KUKA KRL program: MyProgram_087().src

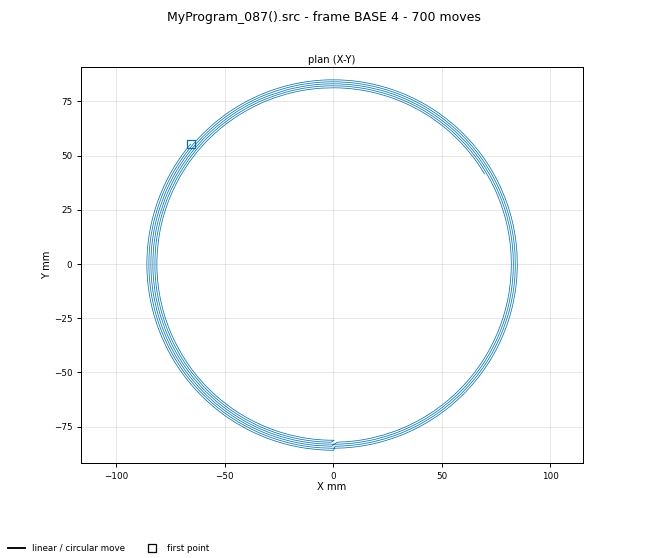
[picture p0: tool path of MyProgram_087().src in frame BASE 4, 700 of 700 moves have a stored position in this frame; points joined in program order, loops and branches not executed]
&ACCESS RVP
&REL 1
&PARAM TEMPLATE = C:\KRC\Roboter\Template\vorgabe
&PARAM EDITMASK = *
DEF MyProgram_087()
; ---- Setting reference (Base) ----
$BASE = BASE_DATA[4]

; --------------------------
; ---- Setting tool (TCP) ----
$TOOL = TOOL_DATA[3]
; --------------------------

$VEL.CP = VEL_APROX_PRINT
Startdeposition()
$VEL.CP = VEL_PRINT
LIN {X -65.6493,Y 55.3345,Z 85,A 135.0931,B 24.9031,C -2.2728,E1 24.8765,E2 309.7224} C_DIS
LIN {X -67.6092,Y 52.9216,Z 85,A 137.2051,B 24.9035,C -2.2684,E1 24.8729,E2 307.6109} C_DIS
LIN {X -69.5478,Y 50.3473,Z 85,A 139.3855,B 24.9039,C -2.2635,E1 24.8693,E2 305.4317} C_DIS
LIN {X -71.5517,Y 47.4546,Z 85,A 141.6093,B 24.9047,C -2.2535,E1 24.8658,E2 303.2206} C_DIS
LIN {X -73.3166,Y 44.6791,Z 85,A 143.8272,B 24.9052,C -2.248,E1 24.8625,E2 301.0046} C_DIS
LIN {X -75.0457,Y 41.7097,Z 85,A 146.1939,B 24.9056,C -2.2435,E1 24.8592,E2 298.6364} C_DIS
LIN {X -76.7013,Y 38.583,Z 85,A 148.5855,B 24.9061,C -2.2374,E1 24.8562,E2 296.2465} C_DIS
LIN {X -78.0463,Y 35.7848,Z 85,A 150.7651,B 24.9064,C -2.2343,E1 24.8536,E2 294.0624} C_DIS
LIN {X -79.8151,Y 31.6411,Z 85,A 154.2705,B 24.9059,C -2.2392,E1 24.8499,E2 290.5257} C_DIS
LIN {X -81.0653,Y 28.2839,Z 85,A 156.0322,B 24.908,C -2.2142,E1 24.8483,E2 288.8137} C_DIS
LIN {X -82.0788,Y 25.1926,Z 85,A 158.531,B 24.9078,C -2.2166,E1 24.8462,E2 286.2947} C_DIS
LIN {X -83.1814,Y 21.2698,Z 85,A 160.8924,B 24.9094,C -2.1981,E1 24.8445,E2 283.9638} C_DIS
LIN {X -83.8706,Y 18.3647,Z 85,A 162.9269,B 24.9098,C -2.193,E1 24.8432,E2 281.9297} C_DIS
LIN {X -84.5105,Y 15.1494,Z 85,A 165.1334,B 24.9103,C -2.1866,E1 24.8421,E2 279.7254} C_DIS
LIN {X -84.9815,Y 12.2354,Z 85,A 167.1994,B 24.9106,C -2.183,E1 24.8412,E2 277.6557} C_DIS
LIN {X -85.4194,Y 8.6682,Z 85,A 169.6631,B 24.9111,C -2.1771,E1 24.8404,E2 275.1912} C_DIS
LIN {X -85.7088,Y 5.064,Z 85,A 171.7651,B 24.9124,C -2.1608,E1 24.84,E2 273.1156} C_DIS
LIN {X -85.8246,Y 2.3935,Z 85,A 173.796,B 24.9124,C -2.1619,E1 24.8398,E2 271.0697} C_DIS
LIN {X -85.8549,Y -0.7778,Z 85,A 175.8922,B 24.9129,C -2.1546,E1 24.8398,E2 268.9783} C_DIS
LIN {X -85.7663,Y -3.9684,Z 85,A 178.1489,B 24.9132,C -2.1514,E1 24.84,E2 266.7158} C_DIS
LIN {X -85.5328,Y -7.4731,Z 85,A -179.4836,B 24.9137,C -2.1446,E1 24.8406,E2 264.3502} C_DIS
LIN {X -85.1548,Y -10.9633,Z 85,A -177.1748,B 24.9144,C -2.1363,E1 24.8413,E2 262.0474} C_DIS
LIN {X -84.6385,Y -14.4197,Z 85,A -174.7821,B 24.9149,C -2.1307,E1 24.8424,E2 259.6538} C_DIS
LIN {X -84.1506,Y -17.0373,Z 85,A -173.063,B 24.9154,C -2.1236,E1 24.8433,E2 257.9415} C_DIS
LIN {X -83.4534,Y -20.1765,Z 85,A -170.9028,B 24.9159,C -2.1175,E1 24.8447,E2 255.7833} C_DIS
LIN {X -82.61,Y -23.3907,Z 85,A -168.7117,B 24.9165,C -2.11,E1 24.8463,E2 253.5972} C_DIS
LIN {X -81.3101,Y -27.5722,Z 85,A -165.6983,B 24.917,C -2.1039,E1 24.8488,E2 250.5811} C_DIS
LIN {X -80.4535,Y -29.9829,Z 85,A -163.7906,B 24.917,C -2.1046,E1 24.8507,E2 248.6611} C_DIS
LIN {X -79.1046,Y -33.3765,Z 85,A -161.4857,B 24.9178,C -2.0939,E1 24.8531,E2 246.369} C_DIS
LIN {X -77.6498,Y -36.6364,Z 85,A -159.0613,B 24.9182,C -2.0883,E1 24.856,E2 243.9444} C_DIS
LIN {X -76.0628,Y -39.8249,Z 85,A -156.9851,B 24.9194,C -2.0733,E1 24.8585,E2 241.893} C_DIS
LIN {X -74.7201,Y -42.2926,Z 85,A -154.847,B 24.9192,C -2.0757,E1 24.8615,E2 239.7378} C_DIS
LIN {X -73.1736,Y -44.9144,Z 85,A -152.7759,B 24.9195,C -2.0716,E1 24.8645,E2 237.666} C_DIS
LIN {X -71.3839,Y -47.7089,Z 85,A -150.4876,B 24.9198,C -2.068,E1 24.868,E2 235.3747} C_DIS
LIN {X -69.3777,Y -50.5796,Z 85,A -148.2542,B 24.9205,C -2.0593,E1 24.8716,E2 233.1512} C_DIS
LIN {X -67.3565,Y -53.2413,Z 85,A -146.0514,B 24.9209,C -2.0532,E1 24.8753,E2 230.9526} C_DIS
LIN {X -65.2873,Y -55.7594,Z 85,A -143.9463,B 24.9215,C -2.0461,E1 24.8791,E2 228.8546} C_DIS
LIN {X -63.1419,Y -58.1779,Z 85,A -141.5868,B 24.9215,C -2.0472,E1 24.8835,E2 226.482} C_DIS
LIN {X -60.5197,Y -60.9013,Z 85,A -139.0966,B 24.9219,C -2.0409,E1 24.8884,E2 223.9962} C_DIS
LIN {X -58.0252,Y -63.282,Z 85,A -136.8032,B 24.9223,C -2.0361,E1 24.8931,E2 221.705} C_DIS
LIN {X -55.4826,Y -65.5232,Z 85,A -134.4958,B 24.9225,C -2.033,E1 24.8979,E2 219.3957} C_DIS
LIN {X -52.8303,Y -67.6812,Z 85,A -132.4193,B 24.9233,C -2.0228,E1 24.9024,E2 217.3358} C_DIS
LIN {X -50.6058,Y -69.3586,Z 85,A -130.3248,B 24.923,C -2.0266,E1 24.9072,E2 215.2249} C_DIS
LIN {X -47.7844,Y -71.3328,Z 85,A -128.0592,B 24.9233,C -2.0219,E1 24.9124,E2 212.9629} C_DIS
LIN {X -45.133,Y -73.0392,Z 85,A -125.8563,B 24.9233,C -2.0217,E1 24.9176,E2 210.7534} C_DIS
LIN {X -40.4274,Y -75.7455,Z 85,A -121.6598,B 24.9224,C -2.0342,E1 24.928,E2 206.5152} C_DIS
LIN {X -37.144,Y -77.4071,Z 85,A -120.0392,B 24.9246,C -2.0059,E1 24.9319,E2 204.9577} C_DIS
LIN {X -34.4456,Y -78.6451,Z 85,A -117.8993,B 24.9244,C -2.0085,E1 24.9374,E2 202.8064} C_DIS
LIN {X -31.4797,Y -79.8785,Z 85,A -115.7324,B 24.9244,C -2.0071,E1 24.943,E2 200.638} C_DIS
LIN {X -28.5704,Y -80.9647,Z 85,A -113.6156,B 24.9244,C -2.0067,E1 24.9485,E2 198.518} C_DIS
LIN {X -25.5353,Y -81.9725,Z 85,A -111.4952,B 24.9247,C -2.0046,E1 24.9542,E2 196.3986} C_DIS
LIN {X -22.9181,Y -82.7438,Z 85,A -109.595,B 24.9246,C -2.0059,E1 24.9593,E2 194.4924} C_DIS
LIN {X -19.7547,Y -83.555,Z 85,A -107.4358,B 24.9246,C -2.0041,E1 24.9651,E2 192.3345} C_DIS
LIN {X -15.6717,Y -84.4166,Z 85,A -104.7417,B 24.925,C -2.0001,E1 24.9725,E2 189.6467} C_DIS
LIN {X -12.5082,Y -84.9427,Z 85,A -102.5283,B 24.9249,C -2.0019,E1 24.9786,E2 187.4273} C_DIS
LIN {X -6.7373,Y -85.5929,Z 85,A -99.1371,B 24.926,C -1.9862,E1 24.988,E2 184.071} C_DIS
LIN {X -3.1736,Y -85.8004,Z 85,A -96.2343,B 24.9248,C -2.0028,E1 24.9962,E2 181.1283} C_DIS
LIN {X 0.2479,Y -85.8577,Z 85,A -93.4453,B 24.9235,C -2.0194,E1 25.0041,E2 178.2998} C_DIS
LIN {X 0.2479,Y -85.8577,Z 85,A -93.4453,B 24.9235,C -2.0194,E1 25.0041,E2 178.2998} C_DIS
Enddeposition()
LIN {X 0.5365,Y -84.9273,Z 85,A -93.1479,B 24.9221,C -2.0386,E1 25.005,E2 177.9569} C_DIS
Startdeposition()
$VEL.CP = VEL_PRINT
LIN {X -0.353,Y -84.9359,Z 85,A -96.7334,B 24.929,C -1.9459,E1 24.9944,E2 181.7624} C_DIS
LIN {X -5.9457,Y -84.7284,Z 85,A -99.0371,B 24.9257,C -1.9903,E1 24.9883,E2 183.9613} C_DIS
LIN {X -10.0146,Y -84.3441,Z 85,A -101.4892,B 24.925,C -1.9999,E1 24.9815,E2 186.3921} C_DIS
LIN {X -12.0876,Y -84.0721,Z 85,A -103.4806,B 24.9263,C -1.9825,E1 24.9759,E2 188.4264} C_DIS
LIN {X -15.4591,Y -83.5189,Z 85,A -105.8149,B 24.9263,C -1.9823,E1 24.9694,E2 190.7634} C_DIS
LIN {X -18.4006,Y -82.9197,Z 85,A -107.581,B 24.9257,C -1.991,E1 24.9647,E2 192.511} C_DIS
LIN {X -20.6463,Y -82.3905,Z 85,A -109.6817,B 24.9268,C -1.9755,E1 24.9589,E2 194.6514} C_DIS
LIN {X -24.6804,Y -81.2731,Z 85,A -112.2511,B 24.9261,C -1.985,E1 24.952,E2 197.2025} C_DIS
LIN {X -27.9054,Y -80.2219,Z 85,A -114.4048,B 24.9257,C -1.9908,E1 24.9464,E2 199.3464} C_DIS
LIN {X -31.5185,Y -78.8735,Z 85,A -117.0724,B 24.9257,C -1.9913,E1 24.9394,E2 202.0186} C_DIS
LIN {X -34.387,Y -77.6647,Z 85,A -119.1143,B 24.9254,C -1.9952,E1 24.9342,E2 204.0559} C_DIS
LIN {X -37.47,Y -76.2252,Z 85,A -121.8843,B 24.9262,C -1.9841,E1 24.9271,E2 206.8596} C_DIS
LIN {X -42.911,Y -73.3006,Z 85,A -125.5069,B 24.9246,C -2.0055,E1 24.9184,E2 210.4415} C_DIS
LIN {X -45.7094,Y -71.5883,Z 85,A -127.4702,B 24.9238,C -2.016,E1 24.9137,E2 212.3858} C_DIS
LIN {X -47.6622,Y -70.3031,Z 85,A -129.5782,B 24.9248,C -2.0032,E1 24.9088,E2 214.5315} C_DIS
LIN {X -50.2302,Y -68.4918,Z 85,A -131.9925,B 24.9251,C -1.9984,E1 24.9033,E2 216.9657} C_DIS
LIN {X -53.1184,Y -66.2786,Z 85,A -134.0621,B 24.924,C -2.0137,E1 24.8988,E2 219.0065} C_DIS
LIN {X -55.5704,Y -64.2362,Z 85,A -136.208,B 24.9236,C -2.018,E1 24.8942,E2 221.1505} C_DIS
LIN {X -57.9324,Y -62.1141,Z 85,A -138.3687,B 24.9234,C -2.0217,E1 24.8898,E2 223.311} C_DIS
LIN {X -60.7411,Y -59.371,Z 85,A -140.818,B 24.9225,C -2.0329,E1 24.885,E2 225.744} C_DIS
LIN {X -62.5685,Y -57.4402,Z 85,A -143.2624,B 24.9236,C -2.0185,E1 24.8802,E2 228.2333} C_DIS
LIN {X -65.9427,Y -53.5329,Z 85,A -146.2237,B 24.9219,C -2.0411,E1 24.875,E2 231.1545} C_DIS
LIN {X -67.897,Y -51.0314,Z 85,A -148.3795,B 24.9215,C -2.0458,E1 24.8713,E2 233.3093} C_DIS
LIN {X -70.6126,Y -47.2051,Z 85,A -151.4442,B 24.9207,C -2.0565,E1 24.8664,E2 236.3637} C_DIS
LIN {X -73.0277,Y -43.3726,Z 85,A -154.3157,B 24.9197,C -2.0695,E1 24.8622,E2 239.2187} C_DIS
LIN {X -74.9807,Y -39.9027,Z 85,A -157.1365,B 24.9194,C -2.0729,E1 24.8584,E2 242.0461} C_DIS
LIN {X -75.98,Y -37.9647,Z 85,A -158.8511,B 24.9196,C -2.0703,E1 24.8562,E2 243.7763} C_DIS
LIN {X -77.3687,Y -35.0474,Z 85,A -161.3363,B 24.9198,C -2.068,E1 24.8532,E2 246.2804} C_DIS
LIN {X -78.933,Y -31.3672,Z 85,A -164.1892,B 24.9195,C -2.0715,E1 24.8502,E2 249.1409} C_DIS
LIN {X -80.2911,Y -27.7072,Z 85,A -167.1343,B 24.9195,C -2.0708,E1 24.8475,E2 252.1044} C_DIS
LIN {X -81.4269,Y -24.1634,Z 85,A -168.8871,B 24.9174,C -2.0988,E1 24.8461,E2 253.8004} C_DIS
LIN {X -82.2605,Y -21.1522,Z 85,A -171.0204,B 24.9169,C -2.1045,E1 24.8446,E2 255.9326} C_DIS
LIN {X -83.1881,Y -17.1447,Z 85,A -173.9455,B 24.9166,C -2.1089,E1 24.8428,E2 258.8643} C_DIS
LIN {X -83.6593,Y -14.6784,Z 85,A -175.662,B 24.9162,C -2.1135,E1 24.8419,E2 260.58} C_DIS
LIN {X -84.1818,Y -11.3038,Z 85,A -177.9693,B 24.9157,C -2.1206,E1 24.841,E2 262.8841} C_DIS
LIN {X -84.6052,Y -7.5007,Z 85,A 179.4059,B 24.9151,C -2.1276,E1 24.8403,E2 265.508} C_DIS
LIN {X -84.7879,Y -5.034,Z 85,A 177.7703,B 24.9146,C -2.1338,E1 24.84,E2 267.1386} C_DIS
LIN {X -84.9203,Y -1.658,Z 85,A 175.5344,B 24.9139,C -2.1422,E1 24.8398,E2 269.3679} C_DIS
LIN {X -84.8865,Y 2.9297,Z 85,A 172.2129,B 24.9136,C -2.146,E1 24.84,E2 272.7004} C_DIS
LIN {X -84.6468,Y 7.0133,Z 85,A 169.6641,B 24.9125,C -2.1605,E1 24.8404,E2 275.23} C_DIS
LIN {X -84.3125,Y 10.2846,Z 85,A 167.392,B 24.912,C -2.1661,E1 24.8411,E2 277.5022} C_DIS
LIN {X -83.9048,Y 13.2,Z 85,A 165.3074,B 24.9117,C -2.1697,E1 24.842,E2 279.5905} C_DIS
LIN {X -83.0805,Y 17.6644,Z 85,A 162.5154,B 24.9103,C -2.1867,E1 24.8435,E2 282.3585} C_DIS
LIN {X -82.5476,Y 20.0028,Z 85,A 160.707,B 24.9103,C -2.1867,E1 24.8446,E2 284.1775} C_DIS
LIN {X -81.0132,Y 25.5189,Z 85,A 156.6749,B 24.9097,C -2.1942,E1 24.8478,E2 288.2152} C_DIS
LIN {X -79.098,Y 30.9471,Z 85,A 153.0309,B 24.9082,C -2.2125,E1 24.8512,E2 291.8359} C_DIS
LIN {X -78.0524,Y 33.4972,Z 85,A 150.7435,B 24.9087,C -2.2066,E1 24.8537,E2 294.1503} C_DIS
LIN {X -76.3679,Y 37.1793,Z 85,A 147.8244,B 24.9084,C -2.2096,E1 24.8572,E2 297.078} C_DIS
LIN {X -74.7656,Y 40.3033,Z 85,A 145.8649,B 24.9069,C -2.2275,E1 24.8597,E2 299.0051} C_DIS
LIN {X -73.177,Y 43.1202,Z 85,A 143.6694,B 24.9064,C -2.2334,E1 24.8628,E2 301.198} C_DIS
LIN {X -70.9482,Y 46.6965,Z 85,A 140.868,B 24.9057,C -2.2425,E1 24.867,E2 303.992} C_DIS
LIN {X -69.2232,Y 49.2176,Z 85,A 138.7614,B 24.9053,C -2.2469,E1 24.8703,E2 306.0985} C_DIS
LIN {X -67.3467,Y 51.7555,Z 85,A 136.6237,B 24.9048,C -2.2523,E1 24.8739,E2 308.2334} C_DIS
LIN {X -65.0503,Y 54.6154,Z 85,A 134.0242,B 24.9046,C -2.2553,E1 24.8785,E2 310.838} C_DIS
LIN {X -62.2698,Y 57.7639,Z 85,A 131.1739,B 24.904,C -2.2619,E1 24.8838,E2 313.6851} C_DIS
LIN {X -59.7294,Y 60.3869,Z 85,A 128.5163,B 24.904,C -2.2625,E1 24.8891,E2 316.3526} C_DIS
LIN {X -56.4358,Y 63.4767,Z 85,A 125.4495,B 24.9034,C -2.2689,E1 24.8954,E2 319.4165} C_DIS
LIN {X -53.9595,Y 65.5954,Z 85,A 123.2848,B 24.9029,C -2.2746,E1 24.9001,E2 321.5758} C_DIS
LIN {X -50.0088,Y 68.6539,Z 85,A 120.5799,B 24.9007,C -2.3003,E1 24.9059,E2 324.2293} C_DIS
LIN {X -47.7834,Y 70.221,Z 85,A 118.3868,B 24.9013,C -2.2939,E1 24.911,E2 326.4452} C_DIS
LIN {X -45.8476,Y 71.4997,Z 85,A 116.6471,B 24.9014,C -2.2919,E1 24.9151,E2 328.1952} C_DIS
LIN {X -43.1027,Y 73.1873,Z 85,A 114.6037,B 24.9008,C -2.2996,E1 24.92,E2 330.2267} C_DIS
LIN {X -40.2759,Y 74.7805,Z 85,A 112.3742,B 24.9006,C -2.3022,E1 24.9254,E2 332.4565} C_DIS
LIN {X -37.315,Y 76.302,Z 85,A 109.3549,B 24.9021,C -2.2838,E1 24.9331,E2 335.5273} C_DIS
LIN {X -33.8752,Y 77.8889,Z 85,A 108.0503,B 24.8987,C -2.3233,E1 24.9362,E2 336.7411} C_DIS
LIN {X -29.1434,Y 79.7801,Z 85,A 103.6943,B 24.9006,C -2.3015,E1 24.9477,E2 341.1584} C_DIS
LIN {X -25.7208,Y 80.9496,Z 85,A 101.1347,B 24.9006,C -2.3009,E1 24.9545,E2 343.7241} C_DIS
LIN {X -22.1417,Y 81.9997,Z 85,A 99.1155,B 24.8992,C -2.3179,E1 24.9598,E2 345.7061} C_DIS
LIN {X -18.9518,Y 82.7953,Z 85,A 96.8259,B 24.8992,C -2.3179,E1 24.9661,E2 347.9988} C_DIS
LIN {X -15.708,Y 83.4721,Z 85,A 94.1004,B 24.9003,C -2.3053,E1 24.9736,E2 350.757} C_DIS
LIN {X -12.463,Y 84.0187,Z 85,A 92.5727,B 24.8984,C -2.3271,E1 24.9777,E2 352.2344} C_DIS
LIN {X -8.7606,Y 84.4835,Z 85,A 89.2154,B 24.9004,C -2.3038,E1 24.9872,E2 355.6491} C_DIS
LIN {X -5.0445,Y 84.7873,Z 85,A 87.4462,B 24.8984,C -2.3268,E1 24.992,E2 357.3643} C_DIS
LIN {X -2.1842,Y 84.9088,Z 85,A 85.068,B 24.8995,C -2.3141,E1 24.9987,E2 359.773} C_DIS
LIN {X 2.8444,Y 84.8892,Z 85,A 81.9748,B 24.8987,C -2.3235,E1 25.0072,E2 362.8435} C_DIS
LIN {X 6.792,Y 84.6645,Z 85,A 79.3621,B 24.8986,C -2.3251,E1 25.0145,E2 365.4512} C_DIS
LIN {X 9.7249,Y 84.378,Z 85,A 77.5037,B 24.8982,C -2.3288,E1 25.0196,E2 367.2997} C_DIS
LIN {X 12.4719,Y 84.0174,Z 85,A 75.4607,B 24.8988,C -2.323,E1 25.0253,E2 369.3547} C_DIS
LIN {X 15.6194,Y 83.4891,Z 85,A 73.3182,B 24.8988,C -2.3225,E1 25.0312,E2 371.496} C_DIS
LIN {X 18.7968,Y 82.8311,Z 85,A 71.1424,B 24.8988,C -2.3219,E1 25.0371,E2 373.6704} C_DIS
LIN {X 22.0041,Y 82.0368,Z 85,A 68.9942,B 24.8988,C -2.323,E1 25.0429,E2 375.8126} C_DIS
LIN {X 24.8674,Y 81.2152,Z 85,A 66.9558,B 24.899,C -2.3207,E1 25.0484,E2 377.8531} C_DIS
LIN {X 28.5484,Y 79.9962,Z 85,A 64.2889,B 24.8993,C -2.3169,E1 25.0555,E2 380.5238} C_DIS
LIN {X 31.9037,Y 78.717,Z 85,A 62.0273,B 24.8991,C -2.3195,E1 25.0613,E2 382.774} C_DIS
LIN {X 33.9922,Y 77.8379,Z 85,A 60.3176,B 24.8997,C -2.3122,E1 25.0657,E2 384.4971} C_DIS
LIN {X 37.9704,Y 75.9772,Z 85,A 57.0434,B 24.9008,C -2.2989,E1 25.074,E2 387.7943} C_DIS
LIN {X 41.2152,Y 74.2668,Z 85,A 54.8695,B 24.9003,C -2.3049,E1 25.0793,E2 389.9474} C_DIS
LIN {X 44.1318,Y 72.5712,Z 85,A 52.6617,B 24.9004,C -2.3038,E1 25.0846,E2 392.1511} C_DIS
LIN {X 47.2175,Y 70.6041,Z 85,A 49.9122,B 24.9015,C -2.2909,E1 25.0911,E2 394.922} C_DIS
LIN {X 51.2507,Y 67.7322,Z 85,A 46.5323,B 24.9021,C -2.2839,E1 25.0987,E2 398.3065} C_DIS
LIN {X 54.8295,Y 64.8694,Z 85,A 43.8514,B 24.9015,C -2.2913,E1 25.1044,E2 400.9598} C_DIS
LIN {X 57.0402,Y 62.935,Z 85,A 41.7448,B 24.9022,C -2.2833,E1 25.1088,E2 403.0768} C_DIS
LIN {X 59.4542,Y 60.659,Z 85,A 39.2032,B 24.9034,C -2.2689,E1 25.1139,E2 405.6419} C_DIS
LIN {X 62.8076,Y 57.1798,Z 85,A 36.4054,B 24.9028,C -2.2767,E1 25.1192,E2 408.409} C_DIS
LIN {X 64.7267,Y 54.997,Z 85,A 34.3639,B 24.9034,C -2.2696,E1 25.123,E2 410.4581} C_DIS
LIN {X 66.8021,Y 52.4571,Z 85,A 32.2778,B 24.9034,C -2.2685,E1 25.1266,E2 412.537} C_DIS
LIN {X 68.818,Y 49.7848,Z 85,A 30.1679,B 24.9035,C -2.2679,E1 25.1301,E2 414.6383} C_DIS
LIN {X 70.365,Y 47.5707,Z 85,A 27.5641,B 24.9061,C -2.2377,E1 25.1343,E2 417.3007} C_DIS
LIN {X 72.3254,Y 44.5364,Z 85,A 25.9399,B 24.9044,C -2.258,E1 25.1366,E2 418.8686} C_DIS
LIN {X 73.7029,Y 42.2149,Z 85,A 23.8817,B 24.9054,C -2.2453,E1 25.1395,E2 420.9461} C_DIS
LIN {X 75.4082,Y 39.0902,Z 85,A 21.0894,B 24.9071,C -2.2259,E1 25.1432,E2 423.7697} C_DIS
LIN {X 77.0939,Y 35.6479,Z 85,A 18.9058,B 24.9066,C -2.2319,E1 25.1458,E2 425.9271} C_DIS
LIN {X 79.4097,Y 30.1382,Z 85,A 15.2343,B 24.9066,C -2.2324,E1 25.1497,E2 429.5774} C_DIS
LIN {X 80.4528,Y 27.2316,Z 85,A 13.2177,B 24.9068,C -2.2285,E1 25.1516,E2 431.5919} C_DIS
LIN {X 81.1497,Y 25.0787,Z 85,A 11.4556,B 24.9079,C -2.216,E1 25.1531,E2 433.3734} C_DIS
LIN {X 82.1086,Y 21.7383,Z 85,A 8.9805,B 24.9088,C -2.2045,E1 25.1549,E2 435.8615} C_DIS
LIN {X 82.8693,Y 18.6314,Z 85,A 6.8379,B 24.9093,C -2.1984,E1 25.1563,E2 438.006} C_DIS
LIN {X 83.5397,Y 15.3436,Z 85,A 4.654,B 24.9097,C -2.1941,E1 25.1574,E2 440.1873} C_DIS
LIN {X 84.0681,Y 12.1155,Z 85,A 2.4566,B 24.9102,C -2.1875,E1 25.1584,E2 442.3874} C_DIS
LIN {X 84.4829,Y 8.7663,Z 85,A -0.2334,B 24.912,C -2.1665,E1 25.1592,E2 445.1111} C_DIS
LIN {X 84.7916,Y 4.9662,Z 85,A -3.6388,B 24.9149,C -2.1306,E1 25.1598,E2 448.5811} C_DIS
LIN {X 84.9334,Y -0.8051,Z 85,A -6.7036,B 24.9136,C -2.1457,E1 25.1598,E2 451.592} C_DIS
LIN {X 84.727,Y -5.9659,Z 85,A -9.7122,B 24.9133,C -2.1505,E1 25.1593,E2 454.5712} C_DIS
LIN {X 84.3693,Y -9.7995,Z 85,A -11.7954,B 24.9125,C -2.1596,E1 25.1587,E2 456.6206} C_DIS
LIN {X 83.9573,Y -12.8603,Z 85,A -14.6434,B 24.9151,C -2.1271,E1 25.1576,E2 459.5286} C_DIS
LIN {X 83.1503,Y -17.329,Z 85,A -17.3155,B 24.9149,C -2.1306,E1 25.1562,E2 462.177} C_DIS
LIN {X 82.486,Y -20.2554,Z 85,A -19.2976,B 24.9153,C -2.1256,E1 25.1549,E2 464.1593} C_DIS
LIN {X 81.5914,Y -23.6064,Z 85,A -21.4994,B 24.9155,C -2.1229,E1 25.1533,E2 466.3548} C_DIS
LIN {X 80.5254,Y -27.0163,Z 85,A -23.864,B 24.916,C -2.1169,E1 25.1513,E2 468.7201} C_DIS
LIN {X 79.6081,Y -29.6143,Z 85,A -25.9992,B 24.9171,C -2.1018,E1 25.1492,E2 470.8789} C_DIS
LIN {X 78.3184,Y -32.8702,Z 85,A -28.2182,B 24.9173,C -2.0995,E1 25.1469,E2 473.0912} C_DIS
LIN {X 77.105,Y -35.6242,Z 85,A -30.4631,B 24.9184,C -2.0862,E1 25.1443,E2 475.3554} C_DIS
LIN {X 75.272,Y -39.3496,Z 85,A -32.8477,B 24.9179,C -2.0919,E1 25.1413,E2 477.7137} C_DIS
LIN {X 74.0505,Y -41.6026,Z 85,A -35.3123,B 24.9202,C -2.0623,E1 25.1379,E2 480.2355} C_DIS
LIN {X 72.384,Y -44.44,Z 85,A -37.4799,B 24.9206,C -2.0577,E1 25.1347,E2 482.4029} C_DIS
LIN {X 69.5014,Y -48.8252,Z 85,A -41.1552,B 24.9217,C -2.0434,E1 25.1289,E2 486.0938} C_DIS
LIN {X 67.3676,Y -51.7284,Z 85,A -42.8343,B 24.9203,C -2.0618,E1 25.1262,E2 487.7213} C_DIS
LIN {X 64.2188,Y -55.5903,Z 85,A -46.0102,B 24.9205,C -2.0592,E1 25.1206,E2 490.8888} C_DIS
LIN {X 61.7492,Y -58.3204,Z 85,A -48.7204,B 24.9215,C -2.0455,E1 25.1154,E2 493.6195} C_DIS
LIN {X 59.027,Y -61.0739,Z 85,A -51.8244,B 24.9233,C -2.023,E1 25.1091,E2 496.7637} C_DIS
LIN {X 56.2479,Y -63.6446,Z 85,A -53.962,B 24.9227,C -2.0307,E1 25.1048,E2 498.8744} C_DIS
LIN {X 53.7083,Y -65.8005,Z 85,A -56.1228,B 24.9228,C -2.0286,E1 25.1001,E2 501.0319} C_DIS
LIN {X 51.0678,Y -67.8697,Z 85,A -59.0946,B 24.9249,C -2.0007,E1 25.0934,E2 504.0589} C_DIS
LIN {X 47.8795,Y -70.1559,Z 85,A -60.7083,B 24.9228,C -2.029,E1 25.0899,E2 505.6002} C_DIS
LIN {X 43.553,Y -72.9211,Z 85,A -64.4287,B 24.9239,C -2.014,E1 25.081,E2 509.3441} C_DIS
LIN {X 39.5471,Y -75.168,Z 85,A -67.4036,B 24.924,C -2.0126,E1 25.0738,E2 512.3136} C_DIS
LIN {X 36.5252,Y -76.6825,Z 85,A -69.8874,B 24.9248,C -2.0023,E1 25.0675,E2 514.815} C_DIS
LIN {X 33.3126,Y -78.1319,Z 85,A -72.1937,B 24.9249,C -2.0011,E1 25.0616,E2 517.1188} C_DIS
LIN {X 30.1881,Y -79.3908,Z 85,A -74.4092,B 24.925,C -1.9998,E1 25.0558,E2 519.3324} C_DIS
LIN {X 27.2497,Y -80.4467,Z 85,A -76.5157,B 24.9252,C -1.9971,E1 25.0503,E2 521.4411} C_DIS
LIN {X 22.924,Y -81.7848,Z 85,A -79.7748,B 24.926,C -1.9871,E1 25.0415,E2 524.7181} C_DIS
LIN {X 19.7248,Y -82.6154,Z 85,A -81.847,B 24.9258,C -1.9898,E1 25.0359,E2 526.7808} C_DIS
LIN {X 16.5183,Y -83.316,Z 85,A -84.0877,B 24.926,C -1.9871,E1 25.0298,E2 529.0252} C_DIS
LIN {X 11.7206,Y -84.1242,Z 85,A -87.086,B 24.9255,C -1.9936,E1 25.0216,E2 532.0051} C_DIS
LIN {X 9.5315,Y -84.4007,Z 85,A -89.6497,B 24.928,C -1.9593,E1 25.0142,E2 534.6482} C_DIS
LIN {X 5.2115,Y -84.7779,Z 85,A -91.5345,B 24.9257,C -1.9901,E1 25.0092,E2 536.4592} C_DIS
LIN {X 0.5365,Y -84.9273,Z 85,A -93.1455,B 24.9221,C -2.0376,E1 25.0051,E2 537.9569} C_DIS
Enddeposition()
LIN {X 0.5365,Y -84.9273,Z 85,A -93.1455,B 24.9221,C -2.0376,E1 25.0051,E2 537.9569} C_DIS
Startdeposition()
$VEL.CP = VEL_PRINT
LIN {X 0.9916,Y -84.0108,Z 85,A -92.9692,B 24.9213,C -2.0489,E1 25.0056,E2 537.7539} C_DIS
LIN {X 4.4731,Y -83.8963,Z 85,A -91.3383,B 24.923,C -2.0265,E1 25.01,E2 536.1768} C_DIS
LIN {X 9.2961,Y -83.5008,Z 85,A -87.8727,B 24.9225,C -2.0333,E1 25.0197,E2 532.6969} C_DIS
LIN {X 11.4949,Y -83.2258,Z 85,A -86.4603,B 24.9226,C -2.0312,E1 25.0235,E2 531.2907} C_DIS
LIN {X 14.2466,Y -82.7995,Z 85,A -84.2028,B 24.9217,C -2.044,E1 25.0298,E2 529.0053} C_DIS
LIN {X 18.3823,Y -81.9811,Z 85,A -81.5361,B 24.922,C -2.0399,E1 25.0371,E2 526.3517} C_DIS
LIN {X 23.2076,Y -80.747,Z 85,A -77.8282,B 24.9209,C -2.0535,E1 25.0471,E2 522.6175} C_DIS
LIN {X 27.7161,Y -79.312,Z 85,A -75.0637,B 24.9218,C -2.0426,E1 25.0544,E2 519.8842} C_DIS
LIN {X 30.8632,Y -78.1413,Z 85,A -72.7119,B 24.9214,C -2.0477,E1 25.0605,E2 517.5254} C_DIS
LIN {X 33.2239,Y -77.1679,Z 85,A -70.705,B 24.9205,C -2.0588,E1 25.0658,E2 515.4969} C_DIS
LIN {X 38.3215,Y -74.7666,Z 85,A -67.3369,B 24.9212,C -2.0495,E1 25.0741,E2 512.1597} C_DIS
LIN {X 40.7639,Y -73.4638,Z 85,A -64.8744,B 24.9195,C -2.0716,E1 25.0803,E2 509.6521} C_DIS
LIN {X 46.0642,Y -70.2617,Z 85,A -61.09,B 24.92,C -2.0651,E1 25.0892,E2 505.8951} C_DIS
LIN {X 47.8199,Y -69.0786,Z 85,A -58.8133,B 24.9176,C -2.0956,E1 25.0945,E2 503.5542} C_DIS
LIN {X 51.2655,Y -66.5614,Z 85,A -56.8074,B 24.9195,C -2.0717,E1 25.0989,E2 501.612} C_DIS
LIN {X 54.8982,Y -63.6003,Z 85,A -53.7778,B 24.9194,C -2.0732,E1 25.1054,E2 498.5904} C_DIS
LIN {X 59.0089,Y -59.8041,Z 85,A -50.0937,B 24.919,C -2.0778,E1 25.1129,E2 494.9106} C_DIS
LIN {X 62.5921,Y -56.0428,Z 85,A -46.5377,B 24.9183,C -2.0869,E1 25.1197,E2 491.3484} C_DIS
LIN {X 64.8496,Y -53.4144,Z 85,A -44.0164,B 24.9174,C -2.0983,E1 25.1243,E2 488.8117} C_DIS
LIN {X 66.4809,Y -51.3699,Z 85,A -41.1728,B 24.9142,C -2.1388,E1 25.1293,E2 485.8859} C_DIS
LIN {X 69.2481,Y -47.5761,Z 85,A -38.8716,B 24.9159,C -2.117,E1 25.1328,E2 483.6475} C_DIS
LIN {X 71.5108,Y -44.0993,Z 85,A -35.5201,B 24.9139,C -2.1428,E1 25.1379,E2 480.2521} C_DIS
LIN {X 73.3225,Y -41.0169,Z 85,A -33.737,B 24.9151,C -2.1276,E1 25.1403,E2 478.5142} C_DIS
LIN {X 74.3931,Y -39.0416,Z 85,A -31.7409,B 24.9135,C -2.1478,E1 25.1429,E2 476.4809} C_DIS
LIN {X 77.0098,Y -33.5865,Z 85,A -28.13,B 24.9139,C -2.1426,E1 25.1471,E2 472.9017} C_DIS
LIN {X 78.2622,Y -30.5553,Z 85,A -25.8185,B 24.9131,C -2.152,E1 25.1495,E2 470.5809} C_DIS
LIN {X 80.4149,Y -24.3355,Z 85,A -21.6297,B 24.9128,C -2.1556,E1 25.1532,E2 466.407} C_DIS
LIN {X 81.3495,Y -20.9959,Z 85,A -19.1323,B 24.9119,C -2.1676,E1 25.1551,E2 463.8959} C_DIS
LIN {X 82.1673,Y -17.5288,Z 85,A -16.2892,B 24.9101,C -2.1893,E1 25.1568,E2 461.0179} C_DIS
LIN {X 82.8484,Y -13.9543,Z 85,A -13.5615,B 24.9087,C -2.2057,E1 25.1581,E2 458.2677} C_DIS
LIN {X 83.3765,Y -10.3504,Z 85,A -11.901,B 24.9104,C -2.1855,E1 25.1587,E2 456.6647} C_DIS
LIN {X 83.7942,Y -6.1064,Z 85,A -8.7143,B 24.9089,C -2.2042,E1 25.1595,E2 453.4525} C_DIS
LIN {X 83.9964,Y -1.7966,Z 85,A -5.9086,B 24.9085,C -2.209,E1 25.1598,E2 450.6523} C_DIS
LIN {X 83.8782,Y 4.801,Z 85,A -1.4715,B 24.9075,C -2.2211,E1 25.1594,E2 446.2129} C_DIS
LIN {X 83.5959,Y 8.3913,Z 85,A 1.0033,B 24.9068,C -2.2295,E1 25.1588,E2 443.7329} C_DIS
LIN {X 83.1907,Y 11.7424,Z 85,A 3.2397,B 24.9063,C -2.2345,E1 25.158,E2 441.4979} C_DIS
LIN {X 82.6797,Y 14.9211,Z 85,A 5.4919,B 24.9056,C -2.2433,E1 25.157,E2 439.2383} C_DIS
LIN {X 82.0292,Y 18.1619,Z 85,A 7.7211,B 24.9051,C -2.2494,E1 25.1557,E2 437.0076} C_DIS
LIN {X 81.0657,Y 22.0669,Z 85,A 10.4005,B 24.9046,C -2.2556,E1 25.1538,E2 434.329} C_DIS
LIN {X 80.1991,Y 25.034,Z 85,A 12.4767,B 24.9041,C -2.2608,E1 25.1521,E2 432.2523} C_DIS
LIN {X 78.7036,Y 29.4017,Z 85,A 15.3833,B 24.9041,C -2.262,E1 25.1495,E2 429.3594} C_DIS
LIN {X 77.6435,Y 32.0946,Z 85,A 17.8924,B 24.902,C -2.2856,E1 25.1468,E2 426.8083} C_DIS
LIN {X 76.0075,Y 35.799,Z 85,A 20.4314,B 24.902,C -2.2859,E1 25.1438,E2 424.2823} C_DIS
LIN {X 74.4672,Y 38.9009,Z 85,A 22.7281,B 24.9016,C -2.2902,E1 25.1409,E2 421.9877} C_DIS
LIN {X 72.9514,Y 41.6739,Z 85,A 25.2285,B 24.9001,C -2.3075,E1 25.1375,E2 419.4593} C_DIS
LIN {X 70.2155,Y 46.1342,Z 85,A 28.6725,B 24.8997,C -2.3126,E1 25.1323,E2 416.0207} C_DIS
LIN {X 67.8324,Y 49.5715,Z 85,A 31.2594,B 24.8998,C -2.3109,E1 25.1281,E2 413.4505} C_DIS
LIN {X 65.8478,Y 52.179,Z 85,A 33.4781,B 24.8994,C -2.3157,E1 25.1243,E2 411.2308} C_DIS
LIN {X 63.732,Y 54.744,Z 85,A 35.7643,B 24.8989,C -2.3215,E1 25.1202,E2 408.9413} C_DIS
LIN {X 61.4628,Y 57.2803,Z 85,A 38.6982,B 24.8967,C -2.3468,E1 25.1146,E2 405.9604} C_DIS
LIN {X 58.8678,Y 59.9434,Z 85,A 40.5918,B 24.898,C -2.3311,E1 25.1109,E2 404.112} C_DIS
LIN {X 55.8178,Y 62.7936,Z 85,A 43.4223,B 24.8976,C -2.3362,E1 25.1051,E2 401.2808} C_DIS
LIN {X 53.2795,Y 64.9623,Z 85,A 45.4506,B 24.8979,C -2.3325,E1 25.1008,E2 399.2692} C_DIS
LIN {X 49.6905,Y 67.7453,Z 85,A 49.3469,B 24.8952,C -2.3638,E1 25.092,E2 395.3129} C_DIS
LIN {X 46.7526,Y 69.8065,Z 85,A 51.5158,B 24.8956,C -2.3587,E1 25.087,E2 393.1632} C_DIS
LIN {X 43.15,Y 72.0892,Z 85,A 53.8583,B 24.8968,C -2.345,E1 25.0815,E2 390.8606} C_DIS
LIN {X 40.4349,Y 73.6463,Z 85,A 55.9627,B 24.8966,C -2.347,E1 25.0764,E2 388.7577} C_DIS
LIN {X 37.2964,Y 75.2831,Z 85,A 59.0884,B 24.8944,C -2.3727,E1 25.0685,E2 385.5797} C_DIS
LIN {X 32.916,Y 77.2994,Z 85,A 61.5908,B 24.8962,C -2.3515,E1 25.0622,E2 383.1337} C_DIS
LIN {X 29.9014,Y 78.5143,Z 85,A 64.1393,B 24.8951,C -2.3641,E1 25.0556,E2 380.561} C_DIS
LIN {X 25.3314,Y 80.1068,Z 85,A 67.4726,B 24.8948,C -2.3679,E1 25.0467,E2 377.2254} C_DIS
LIN {X 21.9475,Y 81.0979,Z 85,A 69.7164,B 24.8951,C -2.3645,E1 25.0407,E2 374.9932} C_DIS
LIN {X 18.4157,Y 81.9737,Z 85,A 72.4692,B 24.8942,C -2.3742,E1 25.0332,E2 372.2212} C_DIS
LIN {X 14.6485,Y 82.7287,Z 85,A 74.9206,B 24.8946,C -2.3701,E1 25.0265,E2 369.7825} C_DIS
LIN {X 11.3758,Y 83.2428,Z 85,A 77.0911,B 24.8948,C -2.368,E1 25.0205,E2 367.619} C_DIS
LIN {X 8.1811,Y 83.6171,Z 85,A 79.5685,B 24.894,C -2.3769,E1 25.0136,E2 365.122} C_DIS
LIN {X 2.6488,Y 83.9735,Z 85,A 83.2484,B 24.8943,C -2.3738,E1 25.0034,E2 361.4509} C_DIS
LIN {X -1.5108,Y 84.0017,Z 85,A 86.0845,B 24.8943,C -2.3731,E1 24.9954,E2 358.6163} C_DIS
LIN {X -5.0829,Y 83.8626,Z 85,A 88.5649,B 24.8943,C -2.3735,E1 24.9885,E2 356.1343} C_DIS
LIN {X -9.2803,Y 83.5026,Z 85,A 91.3034,B 24.8948,C -2.368,E1 24.9809,E2 353.4073} C_DIS
LIN {X -12.3278,Y 83.1075,Z 85,A 93.9923,B 24.8933,C -2.3843,E1 24.9734,E2 350.6774} C_DIS
LIN {X -15.7392,Y 82.528,Z 85,A 95.7075,B 24.8952,C -2.3634,E1 24.9688,E2 349.0102} C_DIS
LIN {X -18.9913,Y 81.8407,Z 85,A 97.9931,B 24.8953,C -2.362,E1 24.9626,E2 346.7251} C_DIS
LIN {X -22.0769,Y 81.063,Z 85,A 101.0597,B 24.8932,C -2.3862,E1 24.9542,E2 343.5963} C_DIS
LIN {X -26.2618,Y 79.8064,Z 85,A 102.907,B 24.8964,C -2.3496,E1 24.9495,E2 341.8328} C_DIS
LIN {X -31.0136,Y 78.082,Z 85,A 106.8286,B 24.8956,C -2.3588,E1 24.9391,E2 337.8813} C_DIS
LIN {X -34.2359,Y 76.7235,Z 85,A 109.5583,B 24.895,C -2.3653,E1 24.9321,E2 335.1295} C_DIS
LIN {X -37.1927,Y 75.3345,Z 85,A 111.547,B 24.8959,C -2.3548,E1 24.9272,E2 333.1604} C_DIS
LIN {X -40.9123,Y 73.3809,Z 85,A 114.0962,B 24.8972,C -2.341,E1 24.921,E2 330.6371} C_DIS
LIN {X -43.7125,Y 71.7481,Z 85,A 116.3629,B 24.8974,C -2.3386,E1 24.9155,E2 328.3691} C_DIS
LIN {X -46.8948,Y 69.7102,Z 85,A 119.3355,B 24.8968,C -2.3448,E1 24.9085,E2 325.3719} C_DIS
LIN {X -50.9422,Y 66.8105,Z 85,A 122.3989,B 24.8983,C -2.3285,E1 24.9017,E2 322.3366} C_DIS
LIN {X -53.288,Y 64.9551,Z 85,A 124.7454,B 24.8979,C -2.3327,E1 24.8966,E2 319.9713} C_DIS
LIN {X -56.5051,Y 62.1764,Z 85,A 127.3616,B 24.8992,C -2.3182,E1 24.8912,E2 317.3792} C_DIS
LIN {X -60.3508,Y 58.4499,Z 85,A 131.6284,B 24.8984,C -2.3267,E1 24.8827,E2 313.0742} C_DIS
LIN {X -62.8028,Y 55.8075,Z 85,A 133.4818,B 24.9004,C -2.3036,E1 24.8793,E2 311.2675} C_DIS
LIN {X -64.7606,Y 53.5227,Z 85,A 135.5547,B 24.9008,C -2.2989,E1 24.8756,E2 309.1963} C_DIS
LIN {X -66.8136,Y 50.9382,Z 85,A 137.8434,B 24.9013,C -2.294,E1 24.8717,E2 306.9084} C_DIS
LIN {X -68.7381,Y 48.3097,Z 85,A 139.7925,B 24.9024,C -2.2805,E1 24.8685,E2 304.982} C_DIS
LIN {X -70.3446,Y 45.9384,Z 85,A 142.5454,B 24.901,C -2.2971,E1 24.8642,E2 302.1756} C_DIS
LIN {X -72.1137,Y 43.1087,Z 85,A 144.316,B 24.9028,C -2.2768,E1 24.8617,E2 300.4446} C_DIS
LIN {X -73.7738,Y 40.1997,Z 85,A 146.1728,B 24.9043,C -2.2586,E1 24.8592,E2 298.6215} C_DIS
LIN {X -76.0291,Y 35.7527,Z 85,A 149.7039,B 24.9049,C -2.252,E1 24.8548,E2 295.0869} C_DIS
LIN {X -77.62,Y 32.1531,Z 85,A 152.8303,B 24.9045,C -2.256,E1 24.8513,E2 291.9339} C_DIS
LIN {X -80.0436,Y 25.5286,Z 85,A 158.2983,B 24.9043,C -2.2592,E1 24.8463,E2 286.4272} C_DIS
LIN {X -81.1416,Y 21.7858,Z 85,A 160.4962,B 24.906,C -2.2382,E1 24.8447,E2 284.2667} C_DIS
LIN {X -81.8672,Y 18.8767,Z 85,A 163.1165,B 24.9052,C -2.2475,E1 24.8431,E2 281.6087} C_DIS
LIN {X -82.7049,Y 14.7812,Z 85,A 165.4028,B 24.9073,C -2.223,E1 24.8419,E2 279.3675} C_DIS
LIN {X -83.3343,Y 10.6761,Z 85,A 168.0364,B 24.9085,C -2.2085,E1 24.8409,E2 276.7526} C_DIS
LIN {X -83.7004,Y 7.2811,Z 85,A 170.2272,B 24.9094,C -2.1974,E1 24.8403,E2 274.5753} C_DIS
LIN {X -83.9612,Y 3.05,Z 85,A 173.9023,B 24.9084,C -2.2095,E1 24.8398,E2 270.8492} C_DIS
LIN {X -84.0146,Y -0.4903,Z 85,A 175.7276,B 24.9104,C -2.1857,E1 24.8398,E2 269.0697} C_DIS
LIN {X -83.9265,Y -3.8693,Z 85,A 177.8341,B 24.9114,C -2.173,E1 24.84,E2 266.9808} C_DIS
LIN {X -83.6775,Y -7.5282,Z 85,A -179.0526,B 24.9107,C -2.1818,E1 24.8407,E2 263.8279} C_DIS
LIN {X -83.135,Y -12.1341,Z 85,A -176.2182,B 24.9123,C -2.1629,E1 24.8417,E2 261.0217} C_DIS
LIN {X -82.744,Y -14.5638,Z 85,A -174.2201,B 24.912,C -2.1664,E1 24.8427,E2 259.0033} C_DIS
LIN {X -81.3768,Y -20.8897,Z 85,A -170.1577,B 24.9138,C -2.1432,E1 24.8452,E2 254.9724} C_DIS
LIN {X -80.6908,Y -23.4056,Z 85,A -168.1488,B 24.9138,C -2.1442,E1 24.8468,E2 252.9495} C_DIS
LIN {X -79.1061,Y -28.303,Z 85,A -164.9444,B 24.9153,C -2.1254,E1 24.8496,E2 249.7718} C_DIS
LIN {X -77.9998,Y -31.2223,Z 85,A -162.6011,B 24.9153,C -2.1251,E1 24.852,E2 247.4159} C_DIS
LIN {X -76.2812,Y -35.2111,Z 85,A -159.6781,B 24.9161,C -2.1157,E1 24.8553,E2 244.4993} C_DIS
LIN {X -74.8445,Y -38.169,Z 85,A -157.5872,B 24.9169,C -2.1053,E1 24.8579,E2 242.422} C_DIS
LIN {X -72.8702,Y -41.8151,Z 85,A -154.7289,B 24.9174,C -2.0985,E1 24.8617,E2 239.5648} C_DIS
LIN {X -71.8942,Y -43.4721,Z 85,A -153.1218,B 24.917,C -2.1033,E1 24.8641,E2 237.9379} C_DIS
LIN {X -69.8412,Y -46.7013,Z 85,A -149.7435,B 24.9158,C -2.1184,E1 24.8694,E2 234.5068} C_DIS
LIN {X -67.3171,Y -50.2697,Z 85,A -147.6556,B 24.9184,C -2.0859,E1 24.8727,E2 232.4864} C_DIS
LIN {X -65.3198,Y -52.8384,Z 85,A -145.6566,B 24.9193,C -2.0744,E1 24.8761,E2 230.5053} C_DIS
LIN {X -61.8444,Y -56.8669,Z 85,A -141.706,B 24.9193,C -2.0753,E1 24.8834,E2 226.5347} C_DIS
LIN {X -59.8585,Y -58.9537,Z 85,A -139.148,B 24.9182,C -2.0881,E1 24.8885,E2 223.9352} C_DIS
LIN {X -57.2266,Y -61.5134,Z 85,A -137.2622,B 24.92,C -2.0653,E1 24.8923,E2 222.0961} C_DIS
LIN {X -54.8517,Y -63.6403,Z 85,A -135.0305,B 24.9202,C -2.0627,E1 24.897,E2 219.8618} C_DIS
LIN {X -53.067,Y -65.1345,Z 85,A -132.6623,B 24.9187,C -2.0825,E1 24.9022,E2 217.4376} C_DIS
LIN {X -49.7309,Y -67.7157,Z 85,A -130.6937,B 24.9211,C -2.0511,E1 24.9065,E2 215.5368} C_DIS
LIN {X -46.1352,Y -70.2149,Z 85,A -127.921,B 24.922,C -2.04,E1 24.9128,E2 212.781} C_DIS
LIN {X -43.0989,Y -72.1195,Z 85,A -125.3905,B 24.922,C -2.0389,E1 24.9188,E2 210.2453} C_DIS
LIN {X -39.9499,Y -73.9093,Z 85,A -122.4163,B 24.9212,C -2.0503,E1 24.9262,E2 207.2354} C_DIS
LIN {X -35.1142,Y -76.3263,Z 85,A -118.5743,B 24.9212,C -2.0506,E1 24.9359,E2 203.3829} C_DIS
LIN {X -30.9498,Y -78.1072,Z 85,A -115.5386,B 24.9215,C -2.0459,E1 24.9437,E2 200.3515} C_DIS
LIN {X -26.6769,Y -79.6677,Z 85,A -112.7248,B 24.9224,C -2.0347,E1 24.9511,E2 197.5589} C_DIS
LIN {X -23.5493,Y -80.6482,Z 85,A -109.8203,B 24.9209,C -2.0534,E1 24.959,E2 194.6052} C_DIS
LIN {X -19.8377,Y -81.6397,Z 85,A -108.0805,B 24.9231,C -2.0252,E1 24.9635,E2 192.9298} C_DIS
LIN {X -17.0223,Y -82.2729,Z 85,A -105.9854,B 24.9229,C -2.0282,E1 24.9693,E2 190.8252} C_DIS
LIN {X -13.7433,Y -82.8837,Z 85,A -103.6315,B 24.9227,C -2.0298,E1 24.9758,E2 188.465} C_DIS
LIN {X -10.5488,Y -83.3508,Z 85,A -101.5681,B 24.9231,C -2.0251,E1 24.9814,E2 186.4111} C_DIS
LIN {X -7.5142,Y -83.6788,Z 85,A -99.2999,B 24.9227,C -2.0307,E1 24.9878,E2 184.1284} C_DIS
LIN {X -0.673,Y -84.0127,Z 85,A -94.7356,B 24.9229,C -2.0278,E1 25.0005,E2 179.5701} C_DIS
LIN {X -0.673,Y -84.0127,Z 85,A -94.7356,B 24.9229,C -2.0278,E1 25.0005,E2 179.5701} C_DIS
Enddeposition()
LIN {X 0.5224,Y -83.0909,Z 85,A -94.0232,B 24.9219,C -2.0408,E1 25.0026,E2 178.827} C_DIS
Startdeposition()
$VEL.CP = VEL_PRINT
LIN {X -5.3809,Y -82.92,Z 85,A -99.4193,B 24.925,C -2.0004,E1 24.9873,E2 184.3199} C_DIS
LIN {X -10.499,Y -82.4284,Z 85,A -102.5228,B 24.924,C -2.0139,E1 24.9787,E2 187.3931} C_DIS
LIN {X -13.6535,Y -81.9647,Z 85,A -104.7703,B 24.924,C -2.013,E1 24.9725,E2 189.6447} C_DIS
LIN {X -17.9694,Y -81.1283,Z 85,A -107.6156,B 24.9235,C -2.0197,E1 24.9648,E2 192.4774} C_DIS
LIN {X -23.867,Y -79.5931,Z 85,A -111.6267,B 24.9229,C -2.0278,E1 24.954,E2 196.4753} C_DIS
LIN {X -27.2076,Y -78.5142,Z 85,A -115.1329,B 24.9251,C -1.9983,E1 24.9445,E2 200.0581} C_DIS
LIN {X -30.7125,Y -77.2108,Z 85,A -117.6491,B 24.9248,C -2.0026,E1 24.938,E2 202.5696} C_DIS
LIN {X -33.9368,Y -75.8483,Z 85,A -119.0764,B 24.9225,C -2.0334,E1 24.9345,E2 203.927} C_DIS
LIN {X -38.1308,Y -73.8295,Z 85,A -123.4461,B 24.9247,C -2.0043,E1 24.9234,E2 208.3775} C_DIS
LIN {X -41.641,Y -71.9078,Z 85,A -125.1923,B 24.9222,C -2.0367,E1 24.9193,E2 210.0518} C_DIS
LIN {X -44.8439,Y -69.9547,Z 85,A -127.544,B 24.9214,C -2.0471,E1 24.9138,E2 212.3858} C_DIS
LIN {X -47.8074,Y -67.9654,Z 85,A -130.5312,B 24.9223,C -2.0362,E1 24.9068,E2 215.4091} C_DIS
LIN {X -51.4248,Y -65.2697,Z 85,A -133.9673,B 24.9225,C -2.0327,E1 24.8991,E2 218.8661} C_DIS
LIN {X -54.314,Y -62.8874,Z 85,A -136.2541,B 24.9215,C -2.0457,E1 24.8943,E2 221.1308} C_DIS
LIN {X -58.9759,Y -58.5364,Z 85,A -140.5794,B 24.9207,C -2.0566,E1 24.8855,E2 225.4477} C_DIS
LIN {X -61.0258,Y -56.3965,Z 85,A -143.2029,B 24.9216,C -2.0452,E1 24.8805,E2 228.11} C_DIS
LIN {X -64.915,Y -51.8736,Z 85,A -146.5941,B 24.9193,C -2.0743,E1 24.8745,E2 231.4474} C_DIS
LIN {X -69.0915,Y -46.1655,Z 85,A -151.8253,B 24.9191,C -2.0767,E1 24.8659,E2 236.6984} C_DIS
LIN {X -71.2835,Y -42.7029,Z 85,A -155.0007,B 24.9193,C -2.0747,E1 24.8612,E2 239.8949} C_DIS
LIN {X -73.69,Y -38.3999,Z 85,A -157.8091,B 24.9173,C -2.0997,E1 24.8576,E2 242.6585} C_DIS
LIN {X -74.9288,Y -35.9209,Z 85,A -160.6137,B 24.9188,C -2.0812,E1 24.8541,E2 245.5223} C_DIS
LIN {X -76.4832,Y -32.4809,Z 85,A -162.4785,B 24.9167,C -2.1082,E1 24.8521,E2 247.3331} C_DIS
LIN {X -77.4954,Y -29.9878,Z 85,A -164.5539,B 24.9167,C -2.1076,E1 24.8499,E2 249.4214} C_DIS
LIN {X -79.814,Y -23.1214,Z 85,A -169.2274,B 24.9148,C -2.131,E1 24.8459,E2 254.0657} C_DIS
LIN {X -80.8037,Y -19.371,Z 85,A -172.2283,B 24.9148,C -2.1306,E1 24.8438,E2 257.0853} C_DIS
LIN {X -81.578,Y -15.8,Z 85,A -174.8071,B 24.9144,C -2.1367,E1 24.8424,E2 259.6646} C_DIS
LIN {X -82.0908,Y -12.8752,Z 85,A -176.7078,B 24.9135,C -2.147,E1 24.8415,E2 261.5522} C_DIS
LIN {X -82.7499,Y -7.5558,Z 85,A 178.9191,B 24.914,C -2.1409,E1 24.8402,E2 265.9659} C_DIS
LIN {X -83.0004,Y -3.9647,Z 85,A 177.3166,B 24.9115,C -2.1717,E1 24.8399,E2 267.5044} C_DIS
LIN {X -83.0799,Y -1.5373,Z 85,A 174.4358,B 24.9136,C -2.1457,E1 24.8398,E2 270.4648} C_DIS
LIN {X -83.042,Y 2.9736,Z 85,A 172.6539,B 24.91,C -2.1902,E1 24.8399,E2 272.1512} C_DIS
LIN {X -82.7916,Y 7.1,Z 85,A 169.4389,B 24.91,C -2.1897,E1 24.8405,E2 275.3867} C_DIS
LIN {X -82.4972,Y 9.9464,Z 85,A 167.3612,B 24.9098,C -2.1933,E1 24.8411,E2 277.4684} C_DIS
LIN {X -81.802,Y 14.5971,Z 85,A 163.7022,B 24.9098,C -2.1927,E1 24.8428,E2 281.1504} C_DIS
LIN {X -81.0666,Y 18.2496,Z 85,A 161.4536,B 24.9085,C -2.2091,E1 24.8441,E2 283.373} C_DIS
LIN {X -79.9114,Y 22.7776,Z 85,A 157.7721,B 24.9086,C -2.2073,E1 24.8468,E2 287.0803} C_DIS
LIN {X -77.6602,Y 29.5558,Z 85,A 153.9256,B 24.905,C -2.2508,E1 24.8502,E2 290.8448} C_DIS
LIN {X -76.5287,Y 32.3728,Z 85,A 150.7855,B 24.9068,C -2.2295,E1 24.8536,E2 294.0532} C_DIS
LIN {X -74.305,Y 37.1941,Z 85,A 147.2015,B 24.9057,C -2.2424,E1 24.8579,E2 297.626} C_DIS
LIN {X -72.2821,Y 40.9896,Z 85,A 144.0933,B 24.9053,C -2.2472,E1 24.8621,E2 300.739} C_DIS
LIN {X -69.7398,Y 45.1788,Z 85,A 140.6952,B 24.9045,C -2.2562,E1 24.8672,E2 304.133} C_DIS
LIN {X -66.8932,Y 49.295,Z 85,A 137.6832,B 24.9027,C -2.2771,E1 24.872,E2 307.1096} C_DIS
LIN {X -65.0521,Y 51.7002,Z 85,A 135.5112,B 24.9024,C -2.2804,E1 24.8757,E2 309.2841} C_DIS
LIN {X -62.869,Y 54.3351,Z 85,A 133.1406,B 24.9019,C -2.2862,E1 24.88,E2 311.6518} C_DIS
LIN {X -59.7156,Y 57.7815,Z 85,A 129.5474,B 24.9021,C -2.2842,E1 24.8869,E2 315.2655} C_DIS
LIN {X -56.5587,Y 60.8769,Z 85,A 126.8326,B 24.9007,C -2.3002,E1 24.8924,E2 317.9533} C_DIS
LIN {X -54.1438,Y 63.0333,Z 85,A 124.4182,B 24.9007,C -2.3003,E1 24.8975,E2 320.3769} C_DIS
LIN {X -49.6994,Y 66.5933,Z 85,A 120.9682,B 24.8989,C -2.3216,E1 24.905,E2 323.7888} C_DIS
LIN {X -46.0039,Y 69.198,Z 85,A 117.2826,B 24.8997,C -2.3122,E1 24.9135,E2 327.5093} C_DIS
LIN {X -42.8032,Y 71.2228,Z 85,A 114.8975,B 24.8987,C -2.3232,E1 24.9191,E2 329.8757} C_DIS
LIN {X -39.9194,Y 72.8779,Z 85,A 112.1133,B 24.8996,C -2.3137,E1 24.926,E2 332.6906} C_DIS
LIN {X -37.0703,Y 74.3671,Z 85,A 110.621,B 24.8975,C -2.3373,E1 24.9296,E2 334.1308} C_DIS
LIN {X -33.8458,Y 75.8894,Z 85,A 107.92,B 24.8978,C -2.3342,E1 24.9365,E2 336.8457} C_DIS
LIN {X -29.509,Y 77.6779,Z 85,A 104.311,B 24.8983,C -2.3282,E1 24.9459,E2 340.4769} C_DIS
LIN {X -21.3758,Y 80.2982,Z 85,A 99.0115,B 24.8962,C -2.3516,E1 24.9599,E2 345.7301} C_DIS
LIN {X -18.8934,Y 80.9179,Z 85,A 96.7467,B 24.8973,C -2.339,E1 24.9661,E2 348.0278} C_DIS
LIN {X -12.2098,Y 82.1936,Z 85,A 92.3923,B 24.8962,C -2.3522,E1 24.978,E2 352.3554} C_DIS
LIN {X -9.2702,Y 82.5763,Z 85,A 89.789,B 24.8975,C -2.3373,E1 24.9854,E2 354.9957} C_DIS
LIN {X -5.0481,Y 82.9419,Z 85,A 87.3488,B 24.8962,C -2.3524,E1 24.9921,E2 357.401} C_DIS
LIN {X -0.8343,Y 83.0903,Z 85,A 84.4397,B 24.8961,C -2.3532,E1 25.0002,E2 360.3086} C_DIS
LIN {X 2.4533,Y 83.0579,Z 85,A 81.8828,B 24.8968,C -2.345,E1 25.0074,E2 362.8845} C_DIS
LIN {X 7.8867,Y 82.7194,Z 85,A 78.0424,B 24.8971,C -2.3423,E1 25.0181,E2 366.7294} C_DIS
LIN {X 12.2104,Y 82.1935,Z 85,A 75.3811,B 24.8962,C -2.3516,E1 25.0254,E2 369.3662} C_DIS
LIN {X 15.3676,Y 81.6614,Z 85,A 72.8553,B 24.8971,C -2.3414,E1 25.0324,E2 371.9136} C_DIS
LIN {X 20.8688,Y 80.4311,Z 85,A 69.2991,B 24.8965,C -2.3491,E1 25.042,E2 375.4463} C_DIS
LIN {X 24.1326,Y 79.5141,Z 85,A 66.257,B 24.8985,C -2.3263,E1 25.0502,E2 378.5372} C_DIS
LIN {X 27.8106,Y 78.3026,Z 85,A 63.6627,B 24.8985,C -2.3263,E1 25.057,E2 381.1263} C_DIS
LIN {X 31.2371,Y 76.9993,Z 85,A 62.0681,B 24.8962,C -2.3521,E1 25.061,E2 382.6562} C_DIS
LIN {X 33.594,Y 76.0017,Z 85,A 60.0409,B 24.8971,C -2.3421,E1 25.0663,E2 384.7022} C_DIS
LIN {X 39.0428,Y 73.3514,Z 85,A 56.0756,B 24.897,C -2.3435,E1 25.0762,E2 388.6537} C_DIS
LIN {X 42.7802,Y 71.2368,Z 85,A 52.3431,B 24.8994,C -2.3154,E1 25.0853,E2 392.4412} C_DIS
LIN {X 45.6444,Y 69.4351,Z 85,A 50.8451,B 24.8975,C -2.3376,E1 25.0887,E2 393.8816} C_DIS
LIN {X 48.4243,Y 67.526,Z 85,A 48.1218,B 24.8989,C -2.3213,E1 25.0949,E2 396.6341} C_DIS
LIN {X 52.2403,Y 64.6188,Z 85,A 45.2156,B 24.8983,C -2.328,E1 25.1013,E2 399.514} C_DIS
LIN {X 54.3055,Y 62.8949,Z 85,A 42.8213,B 24.9001,C -2.3075,E1 25.1065,E2 401.9475} C_DIS
LIN {X 56.995,Y 60.4667,Z 85,A 40.5935,B 24.8998,C -2.3109,E1 25.111,E2 404.158} C_DIS
LIN {X 61.6154,Y 55.7528,Z 85,A 36.3603,B 24.8998,C -2.3112,E1 25.1192,E2 408.3723} C_DIS
LIN {X 63.182,Y 53.9692,Z 85,A 34.5062,B 24.9007,C -2.3006,E1 25.1226,E2 410.2432} C_DIS
LIN {X 65.3177,Y 51.3641,Z 85,A 32.0081,B 24.9017,C -2.2895,E1 25.127,E2 412.7559} C_DIS
LIN {X 67.3673,Y 48.6466,Z 85,A 29.7722,B 24.9018,C -2.2873,E1 25.1307,E2 414.9862} C_DIS
LIN {X 70.0636,Y 44.6742,Z 85,A 26.8045,B 24.9016,C -2.2899,E1 25.1352,E2 417.9329} C_DIS
LIN {X 72.2765,Y 40.9994,Z 85,A 23.8124,B 24.9024,C -2.281,E1 25.1395,E2 420.9308} C_DIS
LIN {X 73.5258,Y 38.7116,Z 85,A 21.5497,B 24.9041,C -2.261,E1 25.1425,E2 423.2288} C_DIS
LIN {X 75.4237,Y 34.8704,Z 85,A 18.9769,B 24.9037,C -2.2652,E1 25.1456,E2 425.7779} C_DIS
LIN {X 77.4392,Y 30.131,Z 85,A 15.6639,B 24.9039,C -2.2628,E1 25.1492,E2 429.0784} C_DIS
LIN {X 79.0046,Y 25.7476,Z 85,A 12.5816,B 24.9044,C -2.2575,E1 25.1521,E2 432.1559} C_DIS
LIN {X 80.0194,Y 22.3965,Z 85,A 9.3269,B 24.9073,C -2.2227,E1 25.1546,E2 435.4741} C_DIS
LIN {X 81.1006,Y 18.0967,Z 85,A 6.7123,B 24.9069,C -2.2278,E1 25.1563,E2 438.0615} C_DIS
LIN {X 81.7683,Y 14.7843,Z 85,A 4.4365,B 24.9074,C -2.2224,E1 25.1575,E2 440.3368} C_DIS
LIN {X 82.3069,Y 11.4138,Z 85,A 2.144,B 24.9078,C -2.217,E1 25.1585,E2 442.6284} C_DIS
LIN {X 82.6507,Y 8.5729,Z 85,A 0.246,B 24.9081,C -2.2133,E1 25.159,E2 444.524} C_DIS
LIN {X 82.9647,Y 4.6358,Z 85,A -3.3036,B 24.9111,C -2.1776,E1 25.1597,E2 448.1369} C_DIS
LIN {X 83.0917,Y 0.713,Z 85,A -4.8033,B 24.9085,C -2.2086,E1 25.1597,E2 449.5544} C_DIS
LIN {X 83.0439,Y -2.9095,Z 85,A -8.2935,B 24.9118,C -2.1679,E1 25.1595,E2 453.1199} C_DIS
LIN {X 82.8598,Y -6.2473,Z 85,A -10.3513,B 24.9118,C -2.1686,E1 25.1591,E2 455.1638} C_DIS
LIN {X 82.4659,Y -10.2091,Z 85,A -13.4799,B 24.9135,C -2.1473,E1 25.1581,E2 458.3243} C_DIS
LIN {X 81.905,Y -14.0109,Z 85,A -15.2318,B 24.9118,C -2.1684,E1 25.1573,E2 460.0162} C_DIS
LIN {X 81.1807,Y -17.7293,Z 85,A -17.8086,B 24.9124,C -2.1612,E1 25.1559,E2 462.5948} C_DIS
LIN {X 80.5834,Y -20.276,Z 85,A -20.521,B 24.9153,C -2.1257,E1 25.154,E2 465.3754} C_DIS
LIN {X 79.5244,Y -24.0985,Z 85,A -23.1027,B 24.9155,C -2.1221,E1 25.1519,E2 467.9507} C_DIS
LIN {X 78.4485,Y -27.3948,Z 85,A -25.274,B 24.9155,C -2.122,E1 25.15,E2 470.1103} C_DIS
LIN {X 77.0226,Y -31.1799,Z 85,A -27.9277,B 24.9159,C -2.1179,E1 25.1473,E2 472.7589} C_DIS
LIN {X 75.3226,Y -35.0877,Z 85,A -30.6193,B 24.9159,C -2.1171,E1 25.1442,E2 475.4376} C_DIS
LIN {X 73.5143,Y -38.7335,Z 85,A -32.8162,B 24.915,C -2.1289,E1 25.1415,E2 477.5949} C_DIS
LIN {X 72.4582,Y -40.6753,Z 85,A -35.8075,B 24.9191,C -2.0766,E1 25.1373,E2 480.6944} C_DIS
LIN {X 70.0976,Y -44.6213,Z 85,A -37.9974,B 24.9173,C -2.0994,E1 25.1341,E2 482.8192} C_DIS
LIN {X 68.282,Y -47.3519,Z 85,A -40.4936,B 24.9184,C -2.0855,E1 25.1301,E2 485.3359} C_DIS
LIN {X 65.9518,Y -50.5474,Z 85,A -43.1219,B 24.9188,C -2.0814,E1 25.1257,E2 487.9615} C_DIS
LIN {X 62.9717,Y -54.2161,Z 85,A -46.0193,B 24.9185,C -2.0846,E1 25.1206,E2 490.8378} C_DIS
LIN {X 60.2281,Y -57.2455,Z 85,A -49.0833,B 24.9197,C -2.0696,E1 25.1148,E2 493.9237} C_DIS
LIN {X 57.3719,Y -60.1087,Z 85,A -52.0822,B 24.9207,C -2.0562,E1 25.1088,E2 496.9419} C_DIS
LIN {X 54.5451,Y -62.6857,Z 85,A -54.7423,B 24.9212,C -2.0494,E1 25.1032,E2 499.6074} C_DIS
LIN {X 50.8603,Y -65.7107,Z 85,A -58.2655,B 24.9224,C -2.0348,E1 25.0954,E2 503.1521} C_DIS
LIN {X 48.0945,Y -67.7613,Z 85,A -59.7888,B 24.9207,C -2.057,E1 25.0921,E2 504.6174} C_DIS
LIN {X 46.0729,Y -69.1526,Z 85,A -61.7763,B 24.9216,C -2.0442,E1 25.0875,E2 506.6285} C_DIS
LIN {X 42.39,Y -71.4684,Z 85,A -65.3589,B 24.9235,C -2.0203,E1 25.0788,E2 510.2565} C_DIS
LIN {X 39.1851,Y -73.2762,Z 85,A -67.0741,B 24.9218,C -2.0418,E1 25.0747,E2 511.9159} C_DIS
LIN {X 34.5113,Y -75.5895,Z 85,A -71.4325,B 24.9241,C -2.0122,E1 25.0636,E2 516.3331} C_DIS
LIN {X 31.3425,Y -76.9563,Z 85,A -72.9102,B 24.9222,C -2.0369,E1 25.06,E2 517.7487} C_DIS
LIN {X 29.0964,Y -77.8341,Z 85,A -75.6361,B 24.9249,C -2.0016,E1 25.0526,E2 520.5524} C_DIS
LIN {X 25.2878,Y -79.1534,Z 85,A -77.7484,B 24.9236,C -2.0188,E1 25.0471,E2 522.6199} C_DIS
LIN {X 19.514,Y -80.7705,Z 85,A -81.5416,B 24.9231,C -2.025,E1 25.037,E2 526.3924} C_DIS
LIN {X 16.9245,Y -81.3526,Z 85,A -84.0295,B 24.9248,C -2.0032,E1 25.03,E2 528.9289} C_DIS
LIN {X 12.0922,Y -82.2106,Z 85,A -86.9166,B 24.9238,C -2.0158,E1 25.0222,E2 531.7831} C_DIS
LIN {X 9.0604,Y -82.5997,Z 85,A -89.4995,B 24.925,C -2.0002,E1 25.0149,E2 534.4013} C_DIS
LIN {X 4.2012,Y -82.9887,Z 85,A -92.5705,B 24.9244,C -2.0074,E1 25.0064,E2 537.4537} C_DIS
LIN {X 0.5224,Y -83.0909,Z 85,A -94.0207,B 24.922,C -2.0397,E1 25.0026,E2 538.827} C_DIS
Enddeposition()
LIN {X 0.5224,Y -83.0909,Z 85,A -94.0207,B 24.922,C -2.0397,E1 25.0026,E2 538.827} C_DIS
Startdeposition()
$VEL.CP = VEL_PRINT
LIN {X 1.9162,Y -82.1516,Z 85,A -92.8994,B 24.9204,C -2.0604,E1 25.0058,E2 537.6569} C_DIS
LIN {X 6.5272,Y -81.9133,Z 85,A -89.5862,B 24.9201,C -2.0647,E1 25.0151,E2 534.335} C_DIS
LIN {X 10.3397,Y -81.5201,Z 85,A -87.0538,B 24.9203,C -2.0619,E1 25.0221,E2 531.8109} C_DIS
LIN {X 13.9593,Y -80.9796,Z 85,A -84.6451,B 24.9205,C -2.0594,E1 25.0287,E2 529.4106} C_DIS
LIN {X 17.128,Y -80.369,Z 85,A -82.2533,B 24.92,C -2.0657,E1 25.0353,E2 527.0068} C_DIS
LIN {X 23.5243,Y -78.7339,Z 85,A -77.8779,B 24.9202,C -2.0633,E1 25.0471,E2 522.6438} C_DIS
LIN {X 28.7053,Y -76.996,Z 85,A -74.0372,B 24.9197,C -2.069,E1 25.0573,E2 518.7971} C_DIS
LIN {X 30.5983,Y -76.2647,Z 85,A -71.8072,B 24.9175,C -2.0968,E1 25.0632,E2 516.5065} C_DIS
LIN {X 33.9958,Y -74.8114,Z 85,A -69.5925,B 24.9181,C -2.0892,E1 25.0687,E2 514.3153} C_DIS
LIN {X 37.882,Y -72.9216,Z 85,A -67.1441,B 24.9192,C -2.0761,E1 25.0748,E2 511.9045} C_DIS
LIN {X 41.3759,Y -70.9972,Z 85,A -63.9715,B 24.9178,C -2.0935,E1 25.0826,E2 508.7} C_DIS
LIN {X 44.5292,Y -69.0621,Z 85,A -61.6514,B 24.9181,C -2.0901,E1 25.088,E2 506.3955} C_DIS
LIN {X 46.9128,Y -67.4654,Z 85,A -59.6587,B 24.9178,C -2.0938,E1 25.0926,E2 504.4008} C_DIS
LIN {X 50.4552,Y -64.8599,Z 85,A -55.9565,B 24.9156,C -2.1209,E1 25.101,E2 500.648} C_DIS
LIN {X 53.084,Y -62.726,Z 85,A -54.5343,B 24.9176,C -2.0957,E1 25.1039,E2 499.2908} C_DIS
LIN {X 55.857,Y -60.2707,Z 85,A -50.9334,B 24.9145,C -2.1348,E1 25.1115,E2 495.612} C_DIS
LIN {X 58.5018,Y -57.7056,Z 85,A -48.4773,B 24.9143,C -2.1373,E1 25.1163,E2 493.1604} C_DIS
LIN {X 60.8992,Y -55.1717,Z 85,A -46.5635,B 24.9152,C -2.1264,E1 25.1198,E2 491.2809} C_DIS
LIN {X 63.1432,Y -52.5865,Z 85,A -43.6241,B 24.9132,C -2.1508,E1 25.1252,E2 488.2973} C_DIS
LIN {X 65.4223,Y -49.7243,Z 85,A -41.3622,B 24.9135,C -2.148,E1 25.129,E2 486.0527} C_DIS
LIN {X 68.1313,Y -45.9407,Z 85,A -38.561,B 24.9139,C -2.1423,E1 25.1334,E2 483.2787} C_DIS
LIN {X 69.9229,Y -43.1668,Z 85,A -35.5269,B 24.9114,C -2.173,E1 25.138,E2 480.1873} C_DIS
LIN {X 71.7986,Y -39.9671,Z 85,A -33.7028,B 24.9129,C -2.1552,E1 25.1404,E2 478.4147} C_DIS
LIN {X 73.4772,Y -36.7913,Z 85,A -30.8518,B 24.9113,C -2.1741,E1 25.1441,E2 475.5344} C_DIS
LIN {X 75.8832,Y -31.5326,Z 85,A -27.1096,B 24.9111,C -2.1766,E1 25.1483,E2 471.8068} C_DIS
LIN {X 77.2007,Y -28.1503,Z 85,A -23.9008,B 24.9086,C -2.207,E1 25.1514,E2 468.5441} C_DIS
LIN {X 78.4524,Y -24.4463,Z 85,A -20.8128,B 24.9069,C -2.2276,E1 25.154,E2 465.4249} C_DIS
LIN {X 79.813,Y -19.552,Z 85,A -18.5078,B 24.9094,C -2.1973,E1 25.1555,E2 463.2047} C_DIS
LIN {X 80.5578,Y -16.214,Z 85,A -15.9415,B 24.9083,C -2.2109,E1 25.157,E2 460.6213} C_DIS
LIN {X 81.1484,Y -12.9416,Z 85,A -13.3381,B 24.9069,C -2.2278,E1 25.1582,E2 457.9933} C_DIS
LIN {X 81.7517,Y -8.313,Z 85,A -10.4032,B 24.9069,C -2.2275,E1 25.1592,E2 455.0764} C_DIS
LIN {X 82.0825,Y -3.8687,Z 85,A -7.7275,B 24.9073,C -2.2231,E1 25.1596,E2 452.427} C_DIS
LIN {X 82.1726,Y -0.4429,Z 85,A -5.0388,B 24.9058,C -2.2407,E1 25.1598,E2 449.7128} C_DIS
LIN {X 82.0566,Y 4.3734,Z 85,A -1.6212,B 24.9047,C -2.2533,E1 25.1594,E2 446.2857} C_DIS
LIN {X 81.8505,Y 7.278,Z 85,A 0.3413,B 24.9044,C -2.2575,E1 25.159,E2 444.3251} C_DIS
LIN {X 81.4575,Y 10.8228,Z 85,A 2.7611,B 24.9039,C -2.2631,E1 25.1582,E2 441.9063} C_DIS
LIN {X 80.9606,Y 14.0713,Z 85,A 5.079,B 24.9032,C -2.2711,E1 25.1571,E2 439.5832} C_DIS
LIN {X 80.3153,Y 17.3742,Z 85,A 7.3328,B 24.9029,C -2.2752,E1 25.1559,E2 437.3326} C_DIS
LIN {X 79.523,Y 20.7006,Z 85,A 9.8499,B 24.9019,C -2.2869,E1 25.1542,E2 434.8025} C_DIS
LIN {X 78.8348,Y 23.1841,Z 85,A 11.5404,B 24.9017,C -2.2888,E1 25.1528,E2 433.1173} C_DIS
LIN {X 77.2259,Y 28.0812,Z 85,A 15.0267,B 24.9011,C -2.2958,E1 25.1497,E2 429.6339} C_DIS
LIN {X 75.407,Y 32.6529,Z 85,A 18.3294,B 24.9006,C -2.3015,E1 25.1463,E2 426.3361} C_DIS
LIN {X 74.3034,Y 35.0942,Z 85,A 20.4067,B 24.8996,C -2.3136,E1 25.1438,E2 424.2416} C_DIS
LIN {X 72.4859,Y 38.7094,Z 85,A 23.2234,B 24.8989,C -2.3211,E1 25.1402,E2 421.4219} C_DIS
LIN {X 69.9273,Y 43.1597,Z 85,A 26.4944,B 24.8989,C -2.3206,E1 25.1356,E2 418.169} C_DIS
LIN {X 67.7952,Y 46.437,Z 85,A 29.5106,B 24.8975,C -2.3369,E1 25.1309,E2 415.1293} C_DIS
LIN {X 65.7432,Y 49.2973,Z 85,A 32.3753,B 24.8958,C -2.3562,E1 25.1261,E2 412.2327} C_DIS
LIN {X 63.024,Y 52.7299,Z 85,A 34.957,B 24.8965,C -2.3481,E1 25.1216,E2 409.6821} C_DIS
LIN {X 59.8799,Y 56.2739,Z 85,A 38.6663,B 24.8947,C -2.3685,E1 25.1145,E2 405.941} C_DIS
LIN {X 56.5927,Y 59.5804,Z 85,A 41.4645,B 24.8954,C -2.3607,E1 25.109,E2 403.1729} C_DIS
LIN {X 53.934,Y 61.9963,Z 85,A 43.8389,B 24.8954,C -2.3615,E1 25.1041,E2 400.806} C_DIS
LIN {X 52.1168,Y 63.5332,Z 85,A 45.7465,B 24.8944,C -2.3725,E1 25.0999,E2 398.8797} C_DIS
LIN {X 48.2595,Y 66.5097,Z 85,A 49.4229,B 24.8931,C -2.3873,E1 25.0916,E2 395.1816} C_DIS
LIN {X 44.8576,Y 68.8503,Z 85,A 52.2455,B 24.8928,C -2.39,E1 25.0851,E2 392.3618} C_DIS
LIN {X 41.6354,Y 70.8444,Z 85,A 54.9035,B 24.8924,C -2.3944,E1 25.0787,E2 389.7016} C_DIS
LIN {X 38.5524,Y 72.5685,Z 85,A 57.5897,B 24.8915,C -2.4046,E1 25.0721,E2 386.9989} C_DIS
LIN {X 35.3035,Y 74.2035,Z 85,A 59.0548,B 24.8942,C -2.3745,E1 25.0686,E2 385.6089} C_DIS
LIN {X 31.9185,Y 75.7206,Z 85,A 62.0145,B 24.8929,C -2.3888,E1 25.0609,E2 382.6225} C_DIS
LIN {X 27.8001,Y 77.3285,Z 85,A 64.8884,B 24.8932,C -2.3854,E1 25.0535,E2 379.7631} C_DIS
LIN {X 25.6106,Y 78.0799,Z 85,A 66.9683,B 24.8918,C -2.4009,E1 25.0479,E2 377.6504} C_DIS
LIN {X 22.8463,Y 78.9345,Z 85,A 68.7763,B 24.8923,C -2.3959,E1 25.0431,E2 375.8573} C_DIS
LIN {X 17.6517,Y 80.2548,Z 85,A 72.9492,B 24.8909,C -2.4112,E1 25.0316,E2 371.6541} C_DIS
LIN {X 14.0609,Y 80.9625,Z 85,A 75.0763,B 24.892,C -2.3993,E1 25.0259,E2 369.5576} C_DIS
LIN {X 10.9118,Y 81.446,Z 85,A 77.8233,B 24.8905,C -2.4156,E1 25.0182,E2 366.7742} C_DIS
LIN {X 7.5921,Y 81.8215,Z 85,A 79.6518,B 24.8918,C -2.4009,E1 25.0132,E2 364.9817} C_DIS
LIN {X 4.3821,Y 82.0562,Z 85,A 81.982,B 24.8916,C -2.4035,E1 25.0067,E2 362.6464} C_DIS
LIN {X -0.1538,Y 82.1735,Z 85,A 85.5739,B 24.8905,C -2.4156,E1 24.9966,E2 359.0261} C_DIS
LIN {X -3.5303,Y 82.0971,Z 85,A 87.317,B 24.8922,C -2.3969,E1 24.9918,E2 357.3271} C_DIS
LIN {X -6.9586,Y 81.8788,Z 85,A 90.0933,B 24.8913,C -2.4069,E1 24.984,E2 354.5258} C_DIS
LIN {X -10.216,Y 81.5362,Z 85,A 92.0191,B 24.8923,C -2.3952,E1 24.9788,E2 352.6265} C_DIS
LIN {X -13.5811,Y 81.0429,Z 85,A 94.7837,B 24.8915,C -2.405,E1 24.9711,E2 349.8362} C_DIS
LIN {X -18.5655,Y 80.0482,Z 85,A 97.9745,B 24.8927,C -2.3917,E1 24.9624,E2 346.673} C_DIS
LIN {X -21.8107,Y 79.2264,Z 85,A 101.1424,B 24.8907,C -2.4133,E1 24.9538,E2 343.4489} C_DIS
LIN {X -25.8472,Y 78.0031,Z 85,A 103.2902,B 24.8931,C -2.3872,E1 24.9482,E2 341.3594} C_DIS
LIN {X -31.438,Y 75.9229,Z 85,A 107.3695,B 24.8938,C -2.3793,E1 24.9376,E2 337.2901} C_DIS
LIN {X -34.2687,Y 74.6877,Z 85,A 109.9771,B 24.8929,C -2.3889,E1 24.9309,E2 334.6534} C_DIS
LIN {X -38.3276,Y 72.6869,Z 85,A 112.9403,B 24.8938,C -2.3784,E1 24.9236,E2 331.7071} C_DIS
LIN {X -40.7476,Y 71.3588,Z 85,A 114.6727,B 24.8946,C -2.3697,E1 24.9194,E2 329.9904} C_DIS
LIN {X -45.1099,Y 68.6841,Z 85,A 117.8266,B 24.8962,C -2.3517,E1 24.912,E2 326.8695} C_DIS
LIN {X -47.7143,Y 66.901,Z 85,A 120.54,B 24.8954,C -2.3614,E1 24.9057,E2 324.1238} C_DIS
LIN {X -51.5331,Y 64.0063,Z 85,A 123.7653,B 24.8963,C -2.3511,E1 24.8986,E2 320.9111} C_DIS
LIN {X -53.6864,Y 62.2126,Z 85,A 125.8656,B 24.8963,C -2.3508,E1 24.8941,E2 318.8036} C_DIS
LIN {X -56.0978,Y 60.0458,Z 85,A 128.0757,B 24.8969,C -2.3442,E1 24.8896,E2 316.6} C_DIS
LIN {X -59.0804,Y 57.1132,Z 85,A 131.1463,B 24.8971,C -2.3414,E1 24.8835,E2 313.5232} C_DIS
LIN {X -61.1002,Y 54.9472,Z 85,A 133.0168,B 24.898,C -2.331,E1 24.8801,E2 311.6692} C_DIS
LIN {X -63.057,Y 52.6902,Z 85,A 135.1281,B 24.8984,C -2.3265,E1 24.8762,E2 309.5591} C_DIS
LIN {X -65.1703,Y 50.0524,Z 85,A 137.3966,B 24.8992,C -2.3179,E1 24.8723,E2 307.3003} C_DIS
LIN {X -66.9552,Y 47.6382,Z 85,A 139.863,B 24.8988,C -2.3223,E1 24.8683,E2 304.8116} C_DIS
LIN {X -69.1337,Y 44.4176,Z 85,A 142.7245,B 24.8991,C -2.3188,E1 24.8639,E2 301.944} C_DIS
LIN {X -72.0839,Y 39.4513,Z 85,A 146.9226,B 24.8997,C -2.3118,E1 24.8581,E2 297.7406} C_DIS
LIN {X -74.6123,Y 34.4306,Z 85,A 150.169,B 24.9023,C -2.2823,E1 24.8542,E2 294.5472} C_DIS
LIN {X -75.433,Y 32.5934,Z 85,A 152.4082,B 24.9007,C -2.3003,E1 24.8516,E2 292.2526} C_DIS
LIN {X -76.7577,Y 29.3379,Z 85,A 153.887,B 24.9036,C -2.267,E1 24.8502,E2 290.8449} C_DIS
LIN {X -77.9264,Y 26.075,Z 85,A 156.189,B 24.9045,C -2.2566,E1 24.8481,E2 288.5548} C_DIS
LIN {X -79.314,Y 21.4868,Z 85,A 159.9172,B 24.9045,C -2.2563,E1 24.8451,E2 284.8058} C_DIS
LIN {X -80.0381,Y 18.6094,Z 85,A 162.1008,B 24.9048,C -2.2528,E1 24.8436,E2 282.6178} C_DIS
LIN {X -80.8981,Y 14.4187,Z 85,A 165.7977,B 24.904,C -2.2623,E1 24.8417,E2 278.8763} C_DIS
LIN {X -81.4573,Y 10.8243,Z 85,A 167.4543,B 24.9066,C -2.2309,E1 24.8411,E2 277.2848} C_DIS
LIN {X -81.7587,Y 8.2465,Z 85,A 170.5899,B 24.9042,C -2.2604,E1 24.8402,E2 274.06} C_DIS
LIN {X -82.1032,Y 3.3865,Z 85,A 173.352,B 24.9065,C -2.2325,E1 24.8398,E2 271.3478} C_DIS
LIN {X -82.1416,Y -2.2815,Z 85,A 176.5466,B 24.9092,C -2.1999,E1 24.8398,E2 268.2118} C_DIS
LIN {X -81.9734,Y -5.71,Z 85,A 179.3895,B 24.9089,C -2.2041,E1 24.8403,E2 265.3417} C_DIS
LIN {X -81.6287,Y -9.4355,Z 85,A -177.7648,B 24.909,C -2.2022,E1 24.8411,E2 262.4835} C_DIS
LIN {X -81.1613,Y -12.8583,Z 85,A -174.6025,B 24.908,C -2.2149,E1 24.8426,E2 259.272} C_DIS
LIN {X -80.295,Y -17.4673,Z 85,A -172.7576,B 24.9119,C -2.1667,E1 24.8435,E2 257.5313} C_DIS
LIN {X -79.2178,Y -21.8431,Z 85,A -169.2647,B 24.9119,C -2.1664,E1 24.8459,E2 254.0188} C_DIS
LIN {X -77.4124,Y -27.5654,Z 85,A -164.8332,B 24.9124,C -2.1606,E1 24.8498,E2 249.5758} C_DIS
LIN {X -76.305,Y -30.4988,Z 85,A -162.7179,B 24.9131,C -2.1524,E1 24.8519,E2 247.4683} C_DIS
LIN {X -74.5907,Y -34.4765,Z 85,A -159.5953,B 24.9136,C -2.1466,E1 24.8555,E2 244.3423} C_DIS
LIN {X -73.3886,Y -36.9693,Z 85,A -157.6717,B 24.914,C -2.1411,E1 24.8579,E2 242.4215} C_DIS
LIN {X -70.4273,Y -42.3384,Z 85,A -153.4142,B 24.915,C -2.1292,E1 24.8637,E2 238.1701} C_DIS
LIN {X -68.3522,Y -45.6133,Z 85,A -149.4142,B 24.9126,C -2.1581,E1 24.8701,E2 234.0811} C_DIS
LIN {X -65.0573,Y -50.1991,Z 85,A -146.7886,B 24.9163,C -2.1122,E1 24.8743,E2 231.5524} C_DIS
LIN {X -60.2545,Y -55.8746,Z 85,A -141.6012,B 24.9173,C -2.1005,E1 24.8838,E2 226.3695} C_DIS
LIN {X -58.127,Y -58.085,Z 85,A -138.1066,B 24.9146,C -2.134,E1 24.8909,E2 222.7801} C_DIS
LIN {X -54.0296,Y -61.9128,Z 85,A -136.0462,B 24.9193,C -2.0744,E1 24.8949,E2 220.8536} C_DIS
LIN {X -51.2206,Y -64.257,Z 85,A -132.3041,B 24.9171,C -2.1031,E1 24.9031,E2 217.0291} C_DIS
LIN {X -48.4215,Y -66.3911,Z 85,A -130.5234,B 24.9189,C -2.0798,E1 24.907,E2 215.2976} C_DIS
LIN {X -45.3014,Y -68.5579,Z 85,A -128.2447,B 24.92,C -2.0651,E1 24.9122,E2 213.0462} C_DIS
LIN {X -43.3569,Y -69.8041,Z 85,A -126.0693,B 24.919,C -2.0786,E1 24.9174,E2 210.8316} C_DIS
LIN {X -41.1558,Y -71.1242,Z 85,A -123.915,B 24.9184,C -2.0866,E1 24.9227,E2 208.652} C_DIS
LIN {X -36.4316,Y -73.6555,Z 85,A -120.3687,B 24.9192,C -2.0764,E1 24.9315,E2 205.1204} C_DIS
LIN {X -33.0807,Y -75.2205,Z 85,A -117.7594,B 24.9193,C -2.0744,E1 24.9381,E2 202.5093} C_DIS
LIN {X -30.252,Y -76.402,Z 85,A -115.8418,B 24.92,C -2.0659,E1 24.9431,E2 200.6078} C_DIS
LIN {X -26.436,Y -77.8047,Z 85,A -113.4872,B 24.9212,C -2.0495,E1 24.9492,E2 198.2874} C_DIS
LIN {X -24.3282,Y -78.4891,Z 85,A -110.8973,B 24.9189,C -2.079,E1 24.9563,E2 195.6229} C_DIS
LIN {X -20.8968,Y -79.4712,Z 85,A -109.0491,B 24.9205,C -2.0586,E1 24.9611,E2 193.8205} C_DIS
LIN {X -18.1612,Y -80.1416,Z 85,A -107.3366,B 24.9212,C -2.0502,E1 24.9657,E2 192.1256} C_DIS
LIN {X -15.4056,Y -80.716,Z 85,A -105.2542,B 24.921,C -2.0529,E1 24.9714,E2 190.0344} C_DIS
LIN {X -12.5182,Y -81.2138,Z 85,A -103.0802,B 24.9207,C -2.0562,E1 24.9775,E2 187.8505} C_DIS
LIN {X -9.4842,Y -81.6238,Z 85,A -100.8876,B 24.9207,C -2.0576,E1 24.9835,E2 185.6531} C_DIS
LIN {X -5.0986,Y -82.0158,Z 85,A -97.4165,B 24.9197,C -2.0696,E1 24.9933,E2 182.1521} C_DIS
LIN {X -1.041,Y -82.1677,Z 85,A -95.0398,B 24.9207,C -2.0563,E1 24.9998,E2 179.8068} C_DIS
LIN {X -1.041,Y -82.1677,Z 85,A -95.0398,B 24.9207,C -2.0563,E1 24.9998,E2 179.8068} C_DIS
Enddeposition()
LIN {X 0.4991,Y -81.247,Z 85,A -94.2171,B 24.92,C -2.065,E1 25.0022,E2 178.9635} C_DIS
Startdeposition()
$VEL.CP = VEL_PRINT
LIN {X -1.9588,Y -81.2295,Z 85,A -96.5753,B 24.9215,C -2.046,E1 24.9955,E2 181.3667} C_DIS
LIN {X -4.8156,Y -81.1096,Z 85,A -99.0169,B 24.9225,C -2.0335,E1 24.9886,E2 183.8386} C_DIS
LIN {X -8.6266,Y -80.7927,Z 85,A -101.5396,B 24.9221,C -2.0388,E1 24.9816,E2 186.3502} C_DIS
LIN {X -11.7968,Y -80.3917,Z 85,A -103.7238,B 24.9219,C -2.0412,E1 24.9756,E2 188.5303} C_DIS
LIN {X -14.8828,Y -79.8786,Z 85,A -106.1041,B 24.9222,C -2.0369,E1 24.969,E2 190.9231} C_DIS
LIN {X -19.6079,Y -78.8512,Z 85,A -110.0287,B 24.9232,C -2.0241,E1 24.9582,E2 194.8835} C_DIS
LIN {X -23.0478,Y -77.9143,Z 85,A -111.9707,B 24.9218,C -2.0419,E1 24.9531,E2 196.7864} C_DIS
LIN {X -25.4598,Y -77.1613,Z 85,A -113.527,B 24.9212,C -2.0496,E1 24.949,E2 198.3271} C_DIS
LIN {X -28.748,Y -75.9961,Z 85,A -116.0534,B 24.9212,C -2.0499,E1 24.9424,E2 200.8579} C_DIS
LIN {X -32.1891,Y -74.6043,Z 85,A -118.7155,B 24.9211,C -2.0513,E1 24.9355,E2 203.5228} C_DIS
LIN {X -36.2975,Y -72.6939,Z 85,A -122.3741,B 24.9218,C -2.0422,E1 24.9262,E2 207.2123} C_DIS
LIN {X -40.7636,Y -70.2872,Z 85,A -125.4178,B 24.9203,C -2.0617,E1 24.9189,E2 210.2183} C_DIS
LIN {X -43.4262,Y -68.6747,Z 85,A -127.7932,B 24.9204,C -2.06,E1 24.9132,E2 212.6052} C_DIS
LIN {X -46.636,Y -66.536,Z 85,A -130.4168,B 24.9199,C -2.067,E1 24.9072,E2 215.221} C_DIS
LIN {X -51.4778,Y -62.8654,Z 85,A -134.8169,B 24.9195,C -2.0715,E1 24.8975,E2 219.6266} C_DIS
LIN {X -53.8696,Y -60.8285,Z 85,A -136.7694,B 24.9186,C -2.0828,E1 24.8934,E2 221.5596} C_DIS
LIN {X -57.2477,Y -57.6593,Z 85,A -140.3248,B 24.9187,C -2.0817,E1 24.8862,E2 225.1325} C_DIS
LIN {X -59.444,Y -55.3931,Z 85,A -143.3062,B 24.9199,C -2.0665,E1 24.8804,E2 228.163} C_DIS
LIN {X -62.057,Y -52.4488,Z 85,A -145.077,B 24.9173,C -2.0993,E1 24.8773,E2 229.8636} C_DIS
LIN {X -63.6332,Y -50.5242,Z 85,A -146.9977,B 24.9173,C -2.099,E1 24.8739,E2 231.7939} C_DIS
LIN {X -65.4063,Y -48.2072,Z 85,A -149.8706,B 24.9187,C -2.0826,E1 24.869,E2 234.7199} C_DIS
LIN {X -67.5916,Y -45.0934,Z 85,A -151.8986,B 24.9168,C -2.1064,E1 24.8659,E2 236.7011} C_DIS
LIN {X -69.4744,Y -42.1328,Z 85,A -154.7822,B 24.9171,C -2.1022,E1 24.8616,E2 239.6096} C_DIS
LIN {X -72.4959,Y -36.692,Z 85,A -159.1176,B 24.9161,C -2.1155,E1 24.856,E2 243.9363} C_DIS
LIN {X -74.7581,Y -31.8302,Z 85,A -162.5109,B 24.9144,C -2.1362,E1 24.8521,E2 247.2989} C_DIS
LIN {X -75.9527,Y -28.8624,Z 85,A -164.8199,B 24.914,C -2.1413,E1 24.8498,E2 249.6085} C_DIS
LIN {X -77.5144,Y -24.3611,Z 85,A -168.129,B 24.9131,C -2.1525,E1 24.8468,E2 252.9097} C_DIS
LIN {X -78.4848,Y -21.024,Z 85,A -171.1575,B 24.9137,C -2.1451,E1 24.8445,E2 255.9734} C_DIS
LIN {X -79.6561,Y -16.0269,Z 85,A -174.7054,B 24.9126,C -2.1581,E1 24.8424,E2 259.5114} C_DIS
LIN {X -80.3591,Y -12.018,Z 85,A -177.4335,B 24.9116,C -2.1706,E1 24.8412,E2 262.2258} C_DIS
LIN {X -80.8675,Y -7.9047,Z 85,A 179.0392,B 24.9121,C -2.1645,E1 24.8402,E2 265.7888} C_DIS
LIN {X -81.159,Y -3.9036,Z 85,A 176.9605,B 24.9098,C -2.1924,E1 24.8399,E2 267.8133} C_DIS
LIN {X -81.234,Y -1.7135,Z 85,A 174.8596,B 24.9106,C -2.1833,E1 24.8398,E2 269.9487} C_DIS
LIN {X -81.2358,Y 1.6112,Z 85,A 173.005,B 24.909,C -2.2031,E1 24.8398,E2 271.7671} C_DIS
LIN {X -81.0012,Y 6.3771,Z 85,A 169.2146,B 24.909,C -2.2031,E1 24.8405,E2 275.5804} C_DIS
LIN {X -80.5034,Y 11.0108,Z 85,A 166.0484,B 24.9078,C -2.2166,E1 24.8416,E2 278.7332} C_DIS
LIN {X -79.8452,Y 15.0561,Z 85,A 163.4694,B 24.9064,C -2.2337,E1 24.8429,E2 281.2868} C_DIS
LIN {X -79.1857,Y 18.2066,Z 85,A 161.191,B 24.9058,C -2.2406,E1 24.8442,E2 283.562} C_DIS
LIN {X -78.3728,Y 21.4387,Z 85,A 158.8498,B 24.9052,C -2.2482,E1 24.8459,E2 285.8987} C_DIS
LIN {X -77.0618,Y 25.756,Z 85,A 155.9978,B 24.9036,C -2.2665,E1 24.8482,E2 288.7234} C_DIS
LIN {X -76.217,Y 28.1591,Z 85,A 154.0605,B 24.9035,C -2.2684,E1 24.85,E2 290.6673} C_DIS
LIN {X -74.3314,Y 32.8152,Z 85,A 150.4257,B 24.9028,C -2.2767,E1 24.8539,E2 294.3024} C_DIS
LIN {X -72.4471,Y 36.7873,Z 85,A 147.136,B 24.9024,C -2.281,E1 24.8579,E2 297.5997} C_DIS
LIN {X -70.6674,Y 40.1019,Z 85,A 144.3504,B 24.902,C -2.2852,E1 24.8616,E2 300.3899} C_DIS
LIN {X -68.5277,Y 43.6564,Z 85,A 140.5157,B 24.9033,C -2.2703,E1 24.8674,E2 304.2797} C_DIS
LIN {X -65.9725,Y 47.4295,Z 85,A 138.2312,B 24.9005,C -2.3027,E1 24.871,E2 306.498} C_DIS
LIN {X -63.4062,Y 50.8105,Z 85,A 135.1772,B 24.9,C -2.309,E1 24.8762,E2 309.5514} C_DIS
LIN {X -61.3145,Y 53.3142,Z 85,A 133.006,B 24.8992,C -2.3183,E1 24.8801,E2 311.7104} C_DIS
LIN {X -59.4001,Y 55.4398,Z 85,A 130.9611,B 24.8988,C -2.3226,E1 24.884,E2 313.7541} C_DIS
LIN {X -57.1683,Y 57.7377,Z 85,A 128.7224,B 24.8983,C -2.3286,E1 24.8884,E2 315.9881} C_DIS
LIN {X -55.1042,Y 59.7112,Z 85,A 126.6744,B 24.8979,C -2.3323,E1 24.8925,E2 318.0355} C_DIS
LIN {X -52.7333,Y 61.8147,Z 85,A 124.3749,B 24.8976,C -2.3356,E1 24.8974,E2 320.3361} C_DIS
LIN {X -50.6538,Y 63.5308,Z 85,A 122.314,B 24.8976,C -2.3356,E1 24.9019,E2 322.405} C_DIS
LIN {X -48.7414,Y 65.0087,Z 85,A 120.3027,B 24.8981,C -2.331,E1 24.9064,E2 324.4344} C_DIS
LIN {X -44.8525,Y 67.7505,Z 85,A 116.4892,B 24.8985,C -2.3254,E1 24.9153,E2 328.2737} C_DIS
LIN {X -41.2297,Y 70.0141,Z 85,A 114.749,B 24.8951,C -2.3647,E1 24.9193,E2 329.9257} C_DIS
LIN {X -36.4362,Y 72.6251,Z 85,A 110.3953,B 24.8957,C -2.3575,E1 24.93,E2 334.3088} C_DIS
LIN {X -33.0868,Y 74.2106,Z 85,A 107.9736,B 24.8949,C -2.3667,E1 24.9361,E2 336.7147} C_DIS
LIN {X -30.7885,Y 75.1927,Z 85,A 105.6859,B 24.8959,C -2.3549,E1 24.9421,E2 339.0356} C_DIS
LIN {X -27.2057,Y 76.5624,Z 85,A 103.0692,B 24.8954,C -2.3607,E1 24.949,E2 341.6438} C_DIS
LIN {X -22.1729,Y 78.1678,Z 85,A 99.728,B 24.8941,C -2.3754,E1 24.9578,E2 344.9557} C_DIS
LIN {X -19.1182,Y 78.9707,Z 85,A 97.6516,B 24.8935,C -2.3818,E1 24.9634,E2 347.02} C_DIS
LIN {X -16.1923,Y 79.6221,Z 85,A 95.4608,B 24.8935,C -2.3815,E1 24.9694,E2 349.2143} C_DIS
LIN {X -11.9223,Y 80.3739,Z 85,A 92.1902,B 24.8939,C -2.3777,E1 24.9784,E2 352.497} C_DIS
LIN {X -7.8636,Y 80.8713,Z 85,A 89.3405,B 24.8937,C -2.3802,E1 24.9863,E2 355.3424} C_DIS
LIN {X -4.9569,Y 81.1018,Z 85,A 87.3481,B 24.8935,C -2.3829,E1 24.9918,E2 357.3293} C_DIS
LIN {X 0.5317,Y 81.25,Z 85,A 83.4794,B 24.8934,C -2.3839,E1 25.0027,E2 361.1957} C_DIS
LIN {X 3.4167,Y 81.1799,Z 85,A 81.0548,B 24.8943,C -2.373,E1 25.0095,E2 363.6456} C_DIS
LIN {X 7.2976,Y 80.9236,Z 85,A 77.8784,B 24.8954,C -2.3605,E1 25.0184,E2 366.8501} C_DIS
LIN {X 11.1828,Y 80.4789,Z 85,A 75.8798,B 24.8936,C -2.3816,E1 25.0238,E2 368.7969} C_DIS
LIN {X 13.6467,Y 80.0979,Z 85,A 73.9669,B 24.894,C -2.3765,E1 25.0291,E2 370.7198} C_DIS
LIN {X 17.2697,Y 79.3953,Z 85,A 71.4207,B 24.894,C -2.377,E1 25.036,E2 373.2618} C_DIS
LIN {X 21.8239,Y 78.2667,Z 85,A 68.2292,B 24.8939,C -2.3784,E1 25.0446,E2 376.4451} C_DIS
LIN {X 25.5147,Y 77.1432,Z 85,A 65.5053,B 24.894,C -2.3762,E1 25.0519,E2 379.1692} C_DIS
LIN {X 27.7311,Y 76.3731,Z 85,A 63.7508,B 24.8944,C -2.3718,E1 25.0565,E2 380.9306} C_DIS
LIN {X 30.7652,Y 75.2022,Z 85,A 61.6763,B 24.8941,C -2.376,E1 25.0619,E2 382.9904} C_DIS
LIN {X 33.3809,Y 74.0781,Z 85,A 59.6778,B 24.8942,C -2.3741,E1 25.067,E2 384.9886} C_DIS
LIN {X 35.6286,Y 73.0249,Z 85,A 57.4585,B 24.8957,C -2.3579,E1 25.0726,E2 387.2404} C_DIS
LIN {X 39.935,Y 70.7614,Z 85,A 54.3524,B 24.8952,C -2.363,E1 25.0802,E2 390.3254} C_DIS
LIN {X 42.4811,Y 69.2626,Z 85,A 52.2168,B 24.8956,C -2.3584,E1 25.0853,E2 392.4654} C_DIS
LIN {X 45.2263,Y 67.5025,Z 85,A 49.3862,B 24.8974,C -2.3387,E1 25.092,E2 395.3332} C_DIS
LIN {X 48.0966,Y 65.4872,Z 85,A 46.8545,B 24.8979,C -2.3327,E1 25.0977,E2 397.8702} C_DIS
LIN {X 51.0701,Y 63.1958,Z 85,A 45.3769,B 24.8952,C -2.3635,E1 25.1008,E2 399.2692} C_DIS
LIN {X 54.0909,Y 60.6304,Z 85,A 42.1461,B 24.8968,C -2.3447,E1 25.1077,E2 402.532} C_DIS
LIN {X 56.4825,Y 58.4088,Z 85,A 40.0848,B 24.8966,C -2.3474,E1 25.1118,E2 404.5783} C_DIS
LIN {X 59.4585,Y 55.3777,Z 85,A 36.3427,B 24.8992,C -2.3178,E1 25.1192,E2 408.3742} C_DIS
LIN {X 61.5937,Y 52.9925,Z 85,A 34.7923,B 24.8977,C -2.3346,E1 25.1219,E2 409.8778} C_DIS
LIN {X 64.4949,Y 49.4196,Z 85,A 31.3441,B 24.899,C -2.3206,E1 25.128,E2 413.3431} C_DIS
LIN {X 66.4059,Y 46.8222,Z 85,A 29.1627,B 24.8992,C -2.3179,E1 25.1315,E2 415.5204} C_DIS
LIN {X 68.3351,Y 43.9565,Z 85,A 26.7351,B 24.8997,C -2.312,E1 25.1353,E2 417.9499} C_DIS
LIN {X 69.8086,Y 41.5774,Z 85,A 24.4146,B 24.9011,C -2.2959,E1 25.1386,E2 420.2965} C_DIS
Enddeposition()
END
